	endMainLoop												:	BOOL;					// End of main loop reached
	endSubLoop												:	BOOL;					// End of sub loop reached                                              
	ElementCount											:	DINT;					// No of array elements
	stackCount,left,right,i,j,k								:	DINT;					// running variables 	
	stack													:	ARRAY[1..32] OF UDINT;	// stack size 32 => ~1 Mio elements *)	
	                                					
	pElement_1												:	POINTER TO BYTE;		// Copy Pointer 1		
	pElement_2												:	POINTER TO BYTE;		// Copy Pointer 2
END_VAR
// ends with true in case of no error	                                    					 					
IF SizeOfStruct = 0 OR SizeOfData = 0
	OR pData = 0 OR pCompareElement = 0
THEN               					                                   					
	bySTRING												:= FALSE;
	RETURN;   
ELSE
	bySTRING												:= TRUE;                          					
END_IF                                 					
          
// calculate no. of Elements                                
ElementCount												:= TO_DINT(SizeOfData / SizeOfStruct);   
                              					
// Quicksort                            					
// initial value of array size          					
left 														:= 1;				// first element
right 														:= ElementCount;	// last element 
stackCount 													:= 1;				// running variable 
                                        	
WHILE NOT endMainLoop DO							
	IF left < right THEN                	
		pPivotElement										:= pCompareElement + (SizeOfStruct * TO_UDINT(SHR(right+left,1)));
		i 													:= left -1;
		j 													:= right +1;
		endSubLoop 											:= FALSE;
		REPEAT
			IF SortInverse
			THEN	// sort descending	
				REPEAT	
					i 										:= i+1;	
					pCmpElement								:= pCompareElement + (SizeOfStruct * TO_UDINT(i-1));
					FOR k := 1 TO MAX_STRING_LENGTH DO // Find unequal char
						// element 1,2 to upper char 	https://www.uni-due.de/hummell/infos/ascii/
						IF pCmpElement^[k] = 0 
							AND IgnoreBlank
						THEN
							CompareElement					:= 127;
						ELSE
							CompareElement					:= SEL(pCmpElement^[k] >= 97(*a*)	AND_THEN pCmpElement^[k] <= 122(*z*), 	pCmpElement^[k],pCmpElement^[k] - 32);		// a --> A
						END_IF						
						IF pPivotElement^[k] = 0 
							AND IgnoreBlank
						THEN
							PivotElement					:= 127;
						ELSE
							PivotElement					:= SEL(pPivotElement^[k] >= 97(*a*) AND_THEN pPivotElement^[k] <= 122(*z*), pPivotElement^[k], 	pPivotElement^[k] - 32);// a --> A
						END_IF
						// Find unequal char
						IF CompareElement <> PivotElement
							OR CompareElement = 0
							OR PivotElement = 0
						THEN
							EXIT;
						END_IF
					END_FOR
				UNTIL (CompareElement <= PivotElement) OR NOT (i < right)	END_REPEAT	
				REPEAT	
					j 										:= j-1;	
					pCmpElement								:= pCompareElement + (SizeOfStruct * TO_UDINT(j-1));
					FOR k := 0 TO MAX_STRING_LENGTH DO // Find unequal char
						// element 1,2 to upper char 	https://www.uni-due.de/hummell/infos/ascii/
						IF pCmpElement^[k] = 0 
							AND IgnoreBlank
						THEN
							CompareElement					:= 127;
						ELSE
							CompareElement					:= SEL(pCmpElement^[k] >= 97(*a*)	AND_THEN pCmpElement^[k] <= 122(*z*), 	pCmpElement^[k],pCmpElement^[k] - 32);		// a --> A
						END_IF
						IF pPivotElement^[k] = 0 
							AND IgnoreBlank
						THEN
							PivotElement					:= 127;
						ELSE
							PivotElement					:= SEL(pPivotElement^[k] >= 97(*a*) AND_THEN pPivotElement^[k] <= 122(*z*), pPivotElement^[k], 	pPivotElement^[k] - 32);// a --> A
						END_IF
						// Find unequal char
						IF CompareElement <> PivotElement
							OR CompareElement = 0
							OR PivotElement = 0
						THEN
							EXIT;
						END_IF
					END_FOR
				UNTIL (CompareElement >= PivotElement) OR NOT (j > left)	END_REPEAT		
			ELSE	// sort ascending
				REPEAT	
					i 										:= i+1;
					pCmpElement								:= pCompareElement + (SizeOfStruct * TO_UDINT(i-1));
					FOR k := 0 TO MAX_STRING_LENGTH DO // Find unequal char
						// element 1,2 to upper char 	https://www.uni-due.de/hummell/infos/ascii/
						IF pCmpElement^[k] = 0 
							AND IgnoreBlank
						THEN
							CompareElement					:= 127;
						ELSE
							CompareElement					:= SEL(pCmpElement^[k] >= 97(*a*)	AND_THEN pCmpElement^[k] <= 122(*z*), 	pCmpElement^[k],pCmpElement^[k] - 32);		// a --> A
						END_IF
						IF pPivotElement^[k] = 0 
							AND IgnoreBlank
						THEN
							PivotElement					:= 127;
						ELSE
							PivotElement					:= SEL(pPivotElement^[k] >= 97(*a*) AND_THEN pPivotElement^[k] <= 122(*z*), pPivotElement^[k], 	pPivotElement^[k] - 32);// a --> A
						END_IF
						// Find unequal char
						IF CompareElement <> PivotElement
							OR CompareElement = 0
							OR PivotElement = 0
						THEN
							EXIT;
						END_IF
					END_FOR
				UNTIL (CompareElement >= PivotElement)	OR NOT (i < right)	END_REPEAT;				
				REPEAT	
					j 										:= j-1;	
					pCmpElement								:= pCompareElement + (SizeOfStruct * TO_UDINT(j-1));
					FOR k := 0 TO MAX_STRING_LENGTH DO // Find unequal char
						// element 1,2 to upper char 	https://www.uni-due.de/hummell/infos/ascii/
						IF pCmpElement^[k] = 0 
							AND IgnoreBlank
						THEN	
							CompareElement					:= 127;
						ELSE
							CompareElement					:= SEL(pCmpElement^[k] >= 97(*a*)	AND_THEN pCmpElement^[k] <= 122(*z*), 	pCmpElement^[k],pCmpElement^[k] - 32);		// a --> A
						END_IF
						IF pPivotElement^[k] = 0
							AND IgnoreBlank 
						THEN
							PivotElement					:= 127;
						ELSE
							PivotElement					:= SEL(pPivotElement^[k] >= 97(*a*) AND_THEN pPivotElement^[k] <= 122(*z*), pPivotElement^[k], 	pPivotElement^[k] - 32);// a --> A
						END_IF
						// Find unequal char
						IF CompareElement <> PivotElement
							OR CompareElement = 0
							OR PivotElement = 0
						THEN
							EXIT;
						END_IF
					END_FOR
				UNTIL (CompareElement <= PivotElement) OR NOT (j > left)	END_REPEAT;
			END_IF
			IF i >= j THEN
				endSubLoop									:= TRUE;
			ELSE                    					
				Allocate(SizeOfStruct);
				pElement_1									:= pData + (SizeOfStruct * TO_UDINT(j-1));
				pElement_2									:= pData + (SizeOfStruct * TO_UDINT(i-1));
				
				IF pElement_Tmp = 0 
					OR_ELSE MEMCPY(pElement_Tmp, pElement_1,	SizeOfStruct) = 0
					OR_ELSE MEMCPY(pElement_1,	pElement_2,		SizeOfStruct) = 0
					OR_ELSE MEMCPY(pElement_2,	pElement_Tmp,	SizeOfStruct) = 0
				THEN
					bySTRING								:= FALSE;
					RETURN;	
				END_IF

			END_IF
		UNTIL endSubLoop END_REPEAT;		
		stack[stackCount] 									:= TO_UDINT(right); 	// save right in stack			
		IF stackCount < 32              					
		THEN                            					
			stackCount 										:= stackCount +1;
		ELSE															// Error stack Limit    
			endMainLoop 									:= TRUE;
			bySTRING										:= FALSE;			
		END_IF                          					
		right 												:= MAX(left, i-1);
	ELSE                                
		IF stackCount = 1 THEN          
			endMainLoop 									:= TRUE;
		ELSE                            					
			left 											:= right+1;       
			stackCount 										:= stackCount -1;	// load from stack
			right											:= TO_DINT(stack[stackCount]);
		END_IF
	END_IF
END_WHILE
END_METHOD

METHOD byTIME : BOOL // returns true if sort ends successfully 
VAR_INPUT
	pData													: 	POINTER TO BYTE := 0;	// ADR(Array) 	
	SizeOfData												: 	UDINT := 0;				// SIZEOF(Array)
	pCompareElement											: 	POINTER TO BYTE := 0;	// ADR(Array[1].TIME)		
	SizeOfStruct											: 	UDINT := 0;				// SIZEOF(Array[1]) 	
END_VAR                                                 
VAR        
	pPivotElement											: 	POINTER TO TIME;		// Pivot value
	PivotElement											: 	TIME;					// Pivot value as TIME	
	pCmpElement												:	POINTER TO TIME;		// compare value
	                                					                            	
	endMainLoop												:	BOOL;					// End of main loop reached
	endSubLoop												:	BOOL;					// End of sub loop reached                                              
	ElementCount											:	DINT;					// No of array elements
	stackCount,left,right,i,j								:	DINT;					// running variables 	
	stack													:	ARRAY[1..32] OF UDINT;	// stack size 32 => ~1 Mio elements *)	
	                                					
	pElement_1												:	POINTER TO BYTE;		// Copy Pointer 1		
	pElement_2												:	POINTER TO BYTE;		// Copy Pointer 2
END_VAR
// ends with true in case of no error	                                    					 					
IF SizeOfStruct = 0 OR SizeOfData = 0
	OR pData = 0 OR pCompareElement = 0
THEN               					                                   					
	byTIME													:= FALSE;
	RETURN;   
ELSE
	byTIME													:= TRUE;                          					
END_IF   

// calculate no. of Elements                                
ElementCount												:= TO_DINT(SizeOfData / SizeOfStruct);                                   					
                                        					
// Quicksort                            					
// initial value of array size          					
left 														:= 1;				// first element
right 														:= ElementCount;	// last element 
stackCount 													:= 1;				// running variable 
                                        	
WHILE NOT endMainLoop DO							
	IF left < right THEN                	
		pPivotElement										:= pCompareElement + (SizeOfStruct * TO_UDINT(SHR(right+left,1)));
		PivotElement										:= pPivotElement^;
		i 													:= left -1;
		j 													:= right +1;
		endSubLoop 											:= FALSE;
		REPEAT
			IF SortInverse
			THEN	// sort descending	
				REPEAT	
					i 										:= i+1;	
					pCmpElement								:= pCompareElement + (SizeOfStruct * TO_UDINT(i-1));
				UNTIL (pCmpElement^ <= PivotElement) OR NOT (i < right)	END_REPEAT	
				REPEAT	
					j 										:= j-1;	
					pCmpElement								:= pCompareElement + (SizeOfStruct * TO_UDINT(j-1));
				UNTIL (pCmpElement^ >= PivotElement) OR NOT (j > left)	END_REPEAT		
			ELSE	// sort ascending
				REPEAT	
					i 										:= i+1;
					pCmpElement								:= pCompareElement + (SizeOfStruct * TO_UDINT(i-1));
				UNTIL (pCmpElement^ >= PivotElement)	OR NOT (i < right)	END_REPEAT;				
				REPEAT	
					j 										:= j-1;	
					pCmpElement								:= pCompareElement + (SizeOfStruct * TO_UDINT(j-1));
				UNTIL (pCmpElement^ <= PivotElement) OR NOT (j > left)	END_REPEAT;
			END_IF
			IF i >= j THEN
				endSubLoop									:= TRUE;
			ELSE                    					
				Allocate(SizeOfStruct);
				pElement_1									:= pData + (SizeOfStruct * TO_UDINT(j-1));
				pElement_2									:= pData + (SizeOfStruct * TO_UDINT(i-1));
				
				IF pElement_Tmp = 0 
					OR_ELSE MEMCPY(pElement_Tmp, pElement_1,	SizeOfStruct) = 0
					OR_ELSE MEMCPY(pElement_1,	pElement_2,		SizeOfStruct) = 0
					OR_ELSE MEMCPY(pElement_2,	pElement_Tmp,	SizeOfStruct) = 0
				THEN
					byTIME									:= FALSE;
					RETURN;	
				END_IF

			END_IF
		UNTIL endSubLoop END_REPEAT;		
		stack[stackCount] 									:= TO_UDINT(right); 	// save right in stack			
		IF stackCount < 32              					
		THEN                            					
			stackCount 										:= stackCount +1;
		ELSE															// Error stack Limit    
			endMainLoop 									:= TRUE;
			byTIME											:= FALSE;			
		END_IF                          					
		right 												:= MAX(left, i-1);
	ELSE                                
		IF stackCount = 1 THEN          
			endMainLoop 									:= TRUE;
		ELSE                            					
			left 											:= right+1;       
			stackCount 										:= stackCount -1;	// load from stack
			right											:= TO_DINT(stack[stackCount]);
		END_IF
	END_IF
END_WHILE
END_METHOD

METHOD byUINT : BOOL // returns true if sort ends successfully 
VAR_INPUT
	pData													: 	POINTER TO BYTE := 0;	// ADR(Array) 	
	SizeOfData												: 	UDINT := 0;				// SIZEOF(Array)
	pCompareElement											: 	POINTER TO BYTE := 0;	// ADR(Array[1].UINT)		
	SizeOfStruct											: 	UDINT := 0;				// SIZEOF(Array[1]) 	
END_VAR                                                 
VAR        
	pPivotElement											: 	POINTER TO UINT;		// Pivot value	
	PivotElement											: 	UINT;					// Pivot value as UINT	
	pCmpElement												:	POINTER TO UINT;		// compare value
	                                					                            	
	endMainLoop												:	BOOL;					// End of main loop reached
	endSubLoop												:	BOOL;					// End of sub loop reached                                              
	ElementCount											:	DINT;					// No of array elements
	stackCount,left,right,i,j								:	DINT;					// running variables 	
	stack													:	ARRAY[1..32] OF UDINT;	// stack size 32 => ~1 Mio elements *)	
	                                					
	pElement_1												:	POINTER TO BYTE;		// Copy Pointer 1		
	pElement_2												:	POINTER TO BYTE;		// Copy Pointer 2
END_VAR
// ends with true in case of no error	                                    					 					
IF SizeOfStruct = 0 OR SizeOfData = 0
	OR pData = 0 OR pCompareElement = 0
THEN               					                                   					
	byUINT													:= FALSE;
	RETURN;   
ELSE
	byUINT													:= TRUE;                          					
END_IF     

// calculate no. of Elements                                
ElementCount												:= TO_DINT(SizeOfData / SizeOfStruct);                                 					
                                        					
// Quicksort                            					
// initial value of array size          					
left 														:= 1;				// first element
right 														:= ElementCount;	// last element 
stackCount 													:= 1;				// running variable 
                                        	
WHILE NOT endMainLoop DO							
	IF left < right THEN                	
		pPivotElement										:= pCompareElement + (SizeOfStruct * TO_UDINT(SHR(right+left,1)));
		PivotElement										:= pPivotElement^;
		i 													:= left -1;
		j 													:= right +1;
		endSubLoop 											:= FALSE;
		REPEAT
			IF SortInverse
			THEN	// sort descending	
				REPEAT	
					i 										:= i+1;	
					pCmpElement								:= pCompareElement + (SizeOfStruct * TO_UDINT(i-1));
				UNTIL (pCmpElement^ <= PivotElement) OR NOT (i < right)	END_REPEAT	
				REPEAT	
					j 										:= j-1;	
					pCmpElement								:= pCompareElement + (SizeOfStruct * TO_UDINT(j-1));
				UNTIL (pCmpElement^ >= PivotElement) OR NOT (j > left)	END_REPEAT		
			ELSE	// sort ascending
				REPEAT	
					i 										:= i+1;
					pCmpElement								:= pCompareElement + (SizeOfStruct * TO_UDINT(i-1));
				UNTIL (pCmpElement^ >= PivotElement)	OR NOT (i < right)	END_REPEAT;				
				REPEAT	
					j 										:= j-1;	
					pCmpElement								:= pCompareElement + (SizeOfStruct * TO_UDINT(j-1));
				UNTIL (pCmpElement^ <= PivotElement) OR NOT (j > left)	END_REPEAT;
			END_IF
			IF i >= j THEN
				endSubLoop									:= TRUE;
			ELSE                    					
				Allocate(SizeOfStruct);
				pElement_1									:= pData + (SizeOfStruct * TO_UDINT(j-1));
				pElement_2									:= pData + (SizeOfStruct * TO_UDINT(i-1));
				
				IF pElement_Tmp = 0 
					OR_ELSE MEMCPY(pElement_Tmp, pElement_1,	SizeOfStruct) = 0
					OR_ELSE MEMCPY(pElement_1,	pElement_2,		SizeOfStruct) = 0
					OR_ELSE MEMCPY(pElement_2,	pElement_Tmp,	SizeOfStruct) = 0
				THEN
					byUINT									:= FALSE;
					RETURN;	
				END_IF

			END_IF
		UNTIL endSubLoop END_REPEAT;		
		stack[stackCount] 									:= TO_UDINT(right); 	// save right in stack			
		IF stackCount < 32              					
		THEN                            					
			stackCount 										:= stackCount +1;
		ELSE															// Error stack Limit    
			endMainLoop 									:= TRUE;
			byUINT											:= FALSE;			
		END_IF                          					
		right 												:= MAX(left, i-1);
	ELSE                                
		IF stackCount = 1 THEN          
			endMainLoop 									:= TRUE;
		ELSE                            					
			left 											:= right+1;       
			stackCount 										:= stackCount -1;	// load from stack
			right											:= TO_DINT(stack[stackCount]);
		END_IF
	END_IF
END_WHILE
END_METHOD

METHOD byUSINT : BOOL // returns true if sort ends successfully 
VAR_INPUT
	pData													: 	POINTER TO BYTE := 0;	// ADR(Array) 	
	SizeOfData												: 	UDINT := 0;				// SIZEOF(Array)
	pCompareElement											: 	POINTER TO BYTE := 0;	// ADR(Array[1].USINT)		
	SizeOfStruct											: 	UDINT := 0;				// SIZEOF(Array[1]) 	
END_VAR                                                 
VAR        
	pPivotElement											: 	POINTER TO USINT;		// Pivot value	
	PivotElement											: 	USINT;					// Pivot value as USINT
	pCmpElement												:	POINTER TO USINT;		// compare value
	                                					                            	
	endMainLoop												:	BOOL;					// End of main loop reached
	endSubLoop												:	BOOL;					// End of sub loop reached                                              
	ElementCount											:	DINT;					// No of array elements
	stackCount,left,right,i,j								:	DINT;					// running variables 	
	stack													:	ARRAY[1..32] OF UDINT;	// stack size 32 => ~1 Mio elements *)	
	                                					
	pElement_1												:	POINTER TO BYTE;		// Copy Pointer 1		
	pElement_2												:	POINTER TO BYTE;		// Copy Pointer 2
END_VAR
// ends with true in case of no error	                                    					 					
IF SizeOfStruct = 0 OR SizeOfData = 0
	OR pData = 0 OR pCompareElement = 0
THEN               					                                   					
	byUSINT													:= FALSE;
	RETURN;   
ELSE
	byUSINT													:= TRUE;                          					
END_IF    

// calculate no. of Elements                                
ElementCount												:= TO_DINT(SizeOfData / SizeOfStruct);                               					
                                        					
// Quicksort                            					
// initial value of array size          					
left 														:= 1;				// first element
right 														:= ElementCount;	// last element 
stackCount 													:= 1;				// running variable 
                                        	
WHILE NOT endMainLoop DO							
	IF left < right THEN                	
		pPivotElement										:= pCompareElement + (SizeOfStruct * TO_UDINT(SHR(right+left,1)));
		PivotElement										:= pPivotElement^;
		i 													:= left -1;
		j 													:= right +1;
		endSubLoop 											:= FALSE;
		REPEAT
			IF SortInverse
			THEN	// sort descending	
				REPEAT	
					i 										:= i+1;	
					pCmpElement								:= pCompareElement + (SizeOfStruct * TO_UDINT(i-1));
				UNTIL (pCmpElement^ <= PivotElement) OR NOT (i < right)	END_REPEAT	
				REPEAT	
					j 										:= j-1;	
					pCmpElement								:= pCompareElement + (SizeOfStruct * TO_UDINT(j-1));
				UNTIL (pCmpElement^ >= PivotElement) OR NOT (j > left)	END_REPEAT		
			ELSE	// sort ascending
				REPEAT	
					i 										:= i+1;
					pCmpElement								:= pCompareElement + (SizeOfStruct * TO_UDINT(i-1));
				UNTIL (pCmpElement^ >= PivotElement)	OR NOT (i < right)	END_REPEAT;				
				REPEAT	
					j 										:= j-1;	
					pCmpElement								:= pCompareElement + (SizeOfStruct * TO_UDINT(j-1));
				UNTIL (pCmpElement^ <= PivotElement) OR NOT (j > left)	END_REPEAT;
			END_IF
			IF i >= j THEN
				endSubLoop									:= TRUE;
			ELSE                    					
				Allocate(SizeOfStruct);
				pElement_1									:= pData + (SizeOfStruct * TO_UDINT(j-1));
				pElement_2									:= pData + (SizeOfStruct * TO_UDINT(i-1));
				
				IF pElement_Tmp = 0 
					OR_ELSE MEMCPY(pElement_Tmp, pElement_1,	SizeOfStruct) = 0
					OR_ELSE MEMCPY(pElement_1,	pElement_2,		SizeOfStruct) = 0
					OR_ELSE MEMCPY(pElement_2,	pElement_Tmp,	SizeOfStruct) = 0
				THEN
					byUSINT									:= FALSE;
					RETURN;	
				END_IF

			END_IF
		UNTIL endSubLoop END_REPEAT;		
		stack[stackCount] 									:= TO_UDINT(right); 	// save right in stack			
		IF stackCount < 32              					
		THEN                            					
			stackCount 										:= stackCount +1;
		ELSE															// Error stack Limit    
			endMainLoop 									:= TRUE;
			byUSINT											:= FALSE;			
		END_IF                          					
		right 												:= MAX(left, i-1);
	ELSE                                
		IF stackCount = 1 THEN          
			endMainLoop 									:= TRUE;
		ELSE                            					
			left 											:= right+1;       
			stackCount 										:= stackCount -1;	// load from stack
			right											:= TO_DINT(stack[stackCount]);
		END_IF
	END_IF
END_WHILE
END_METHOD

METHOD byWSTRING : BOOL // returns true if sort ends successfully 
VAR_INPUT
	pData													: 	POINTER TO BYTE := 0;	// ADR(Array) 	
	SizeOfData												: 	UDINT := 0;				// SIZEOF(Array)
	pCompareElement											: 	POINTER TO BYTE := 0;	// ADR(Array[1].WSTRING)		
	SizeOfStruct											: 	UDINT := 0;				// SIZEOF(Array[1]) 	
END_VAR                                                                                            
VAR        
	pPivotElement											: 	POINTER TO WSTRING(MAX_WSTRING_LENGTH);	// Pivot value	
	pCmpElement												:	POINTER TO WSTRING(MAX_WSTRING_LENGTH);	// compare value
	PivotElement											:	WORD; 					// Pivot value	
	CompareElement											:	WORD; 					// compare value
	                                					                            	
	endMainLoop												:	BOOL;					// End of main loop reached
	endSubLoop												:	BOOL;					// End of sub loop reached                                              
	ElementCount											:	DINT;					// No of array elements
	stackCount,left,right,i,j,k								:	DINT;					// running variables 	
	stack													:	ARRAY[1..32] OF UDINT;	// stack size 32 => ~1 Mio elements *)	
	                                					
	pElement_1												:	POINTER TO BYTE;		// Copy Pointer 1		
	pElement_2												:	POINTER TO BYTE;		// Copy Pointer 2
END_VAR
// ends with true in case of no error	                                    					 					
IF SizeOfStruct = 0 OR SizeOfData = 0
	OR pData = 0 OR pCompareElement = 0
THEN               					                                   					
	byWSTRING												:= FALSE;
	RETURN;   
ELSE
	byWSTRING												:= TRUE;                          					
END_IF                                   					
            
// calculate no. of Elements                                
ElementCount												:= TO_DINT(SizeOfData / SizeOfStruct);   
                            					
// Quicksort                            					
// initial value of array size          					
left 														:= 1;				// first element
right 														:= ElementCount;	// last element 
stackCount 													:= 1;				// running variable 
                                        	
WHILE NOT endMainLoop DO							
	IF left < right THEN                	
		pPivotElement										:= pCompareElement + (SizeOfStruct * TO_UDINT(SHR(right+left,1)));
		i 													:= left -1;
		j 													:= right +1;
		endSubLoop 											:= FALSE;
		REPEAT
			IF SortInverse
			THEN	// sort descending	
				REPEAT	
					i 										:= i+1;	
					pCmpElement								:= pCompareElement + (SizeOfStruct * TO_UDINT(i-1));
					FOR k := 0 TO MAX_WSTRING_LENGTH DO // Find unequal char
						// element 1,2 to upper char 	https://www.uni-due.de/hummell/infos/ascii/
						IF pCmpElement^[k] = 0 
							AND IgnoreBlank
						THEN
							CompareElement					:= 127;
						ELSE
							CompareElement					:= SEL(pCmpElement^[k] >= 97(*a*)	AND_THEN pCmpElement^[k] <= 122(*z*), 	pCmpElement^[k],pCmpElement^[k] - 32);		// a --> A
						END_IF
						IF pPivotElement^[k] = 0 
							AND IgnoreBlank
						THEN
							PivotElement					:= 127;
						ELSE
							PivotElement					:= SEL(pPivotElement^[k] >= 97(*a*) AND_THEN pPivotElement^[k] <= 122(*z*), pPivotElement^[k], 	pPivotElement^[k] - 32);// a --> A
						END_IF
						// Find unequal char
						IF CompareElement <> PivotElement
							OR CompareElement = 0
							OR PivotElement = 0
						THEN
							EXIT;
						END_IF
					END_FOR
				UNTIL (CompareElement <= PivotElement) OR NOT (i < right)	END_REPEAT	
				REPEAT	
					j 										:= j-1;	
					pCmpElement								:= pCompareElement + (SizeOfStruct * TO_UDINT(j-1));
					FOR k := 0 TO MAX_WSTRING_LENGTH DO // Find unequal char
						// element 1,2 to upper char 	https://www.uni-due.de/hummell/infos/ascii/
						IF pCmpElement^[k] = 0 
							AND IgnoreBlank
						THEN
							CompareElement					:= 127;
						ELSE
							CompareElement					:= SEL(pCmpElement^[k] >= 97(*a*)	AND_THEN pCmpElement^[k] <= 122(*z*), 	pCmpElement^[k],pCmpElement^[k] - 32);		// a --> A
						END_IF
						IF pPivotElement^[k] = 0 
							AND IgnoreBlank
						THEN
							PivotElement					:= 127;
						ELSE
							PivotElement					:= SEL(pPivotElement^[k] >= 97(*a*) AND_THEN pPivotElement^[k] <= 122(*z*), pPivotElement^[k], 	pPivotElement^[k] - 32);// a --> A
						END_IF
						// Find unequal char
						IF CompareElement <> PivotElement
							OR CompareElement = 0
							OR PivotElement = 0
						THEN
							EXIT;
						END_IF
					END_FOR
				UNTIL (CompareElement >= PivotElement) OR NOT (j > left)	END_REPEAT		
			ELSE	// sort ascending
				REPEAT	
					i 										:= i+1;
					pCmpElement								:= pCompareElement + (SizeOfStruct * TO_UDINT(i-1));
					FOR k := 0 TO MAX_WSTRING_LENGTH DO // Find unequal char
						// element 1,2 to upper char 	https://www.uni-due.de/hummell/infos/ascii/
						IF pCmpElement^[k] = 0 
							AND IgnoreBlank
						THEN
							CompareElement					:= 127;
						ELSE
							CompareElement					:= SEL(pCmpElement^[k] >= 97(*a*)	AND_THEN pCmpElement^[k] <= 122(*z*), 	pCmpElement^[k],pCmpElement^[k] - 32);		// a --> A
						END_IF
						IF pPivotElement^[k] = 0 
							AND IgnoreBlank
						THEN
							PivotElement					:= 127;
						ELSE
							PivotElement					:= SEL(pPivotElement^[k] >= 97(*a*) AND_THEN pPivotElement^[k] <= 122(*z*), pPivotElement^[k], 	pPivotElement^[k] - 32);// a --> A
						END_IF
						// Find unequal char
						IF CompareElement <> PivotElement
							OR CompareElement = 0
							OR PivotElement = 0
						THEN
							EXIT;
						END_IF
					END_FOR
				UNTIL (CompareElement >= PivotElement)	OR NOT (i < right)	END_REPEAT;				
				REPEAT	
					j 										:= j-1;	
					pCmpElement								:= pCompareElement + (SizeOfStruct * TO_UDINT(j-1));
					FOR k := 0 TO MAX_WSTRING_LENGTH DO // Find unequal char
						// element 1,2 to upper char 	https://www.uni-due.de/hummell/infos/ascii/
						IF pCmpElement^[k] = 0 
							AND IgnoreBlank
						THEN
							CompareElement					:= 127;
						ELSE
							CompareElement					:= SEL(pCmpElement^[k] >= 97(*a*)	AND_THEN pCmpElement^[k] <= 122(*z*), 	pCmpElement^[k],pCmpElement^[k] - 32);		// a --> A
						END_IF
						IF pPivotElement^[k] = 0 
							AND IgnoreBlank
						THEN
							PivotElement					:= 127;
						ELSE
							PivotElement					:= SEL(pPivotElement^[k] >= 97(*a*) AND_THEN pPivotElement^[k] <= 122(*z*), pPivotElement^[k], 	pPivotElement^[k] - 32);// a --> A
						END_IF
						// Find unequal char
						IF CompareElement <> PivotElement
							OR CompareElement = 0
							OR PivotElement = 0
						THEN
							EXIT;
						END_IF
					END_FOR
				UNTIL (CompareElement <= PivotElement) OR NOT (j > left)	END_REPEAT;
			END_IF
			IF i >= j THEN
				endSubLoop									:= TRUE;
			ELSE                    					
				Allocate(SizeOfStruct);
				pElement_1									:= pData + (SizeOfStruct * TO_UDINT(j-1));
				pElement_2									:= pData + (SizeOfStruct * TO_UDINT(i-1));
				
				IF pElement_Tmp = 0 
					OR_ELSE MEMCPY(pElement_Tmp, pElement_1,	SizeOfStruct) = 0
					OR_ELSE MEMCPY(pElement_1,	pElement_2,		SizeOfStruct) = 0
					OR_ELSE MEMCPY(pElement_2,	pElement_Tmp,	SizeOfStruct) = 0
				THEN
					byWSTRING								:= FALSE;
					RETURN;	
				END_IF

			END_IF
		UNTIL endSubLoop END_REPEAT;		
		stack[stackCount] 									:= TO_UDINT(right); 	// save right in stack			
		IF stackCount < 32              					
		THEN                            					
			stackCount 										:= stackCount +1;
		ELSE															// Error stack Limit    
			endMainLoop 									:= TRUE;
			byWSTRING										:= FALSE;			
		END_IF                          					
		right 												:= MAX(left, i-1);
	ELSE                                
		IF stackCount = 1 THEN          
			endMainLoop 									:= TRUE;
		ELSE                            					
			left 											:= right+1;       
			stackCount 										:= stackCount -1;	// load from stack
			right											:= TO_DINT(stack[stackCount]);
		END_IF
	END_IF
END_WHILE
END_METHOD

METHOD FB_exit : BOOL
VAR_INPUT
	bInCopyCode : BOOL; // if TRUE, the exit method is called for exiting an instance that is copied afterwards (online change).
END_VAR
IF NOT bInCopyCode AND pElement_Tmp <> 0
THEN //Release memory in case the PLC stopps
	__DELETE(pElement_Tmp);
END_IF
END_METHOD

END_FUNCTION_BLOCK

// ---- POUs/DataBuffer/Ringbuffer/Ringbuffer.TcPOU
//Ringbuffer based on external memory
FUNCTION_BLOCK Ringbuffer EXTENDS RingbufferBase
VAR_INPUT	
END_VAR
VAR_OUTPUT
END_VAR    
VAR
END_VAR

METHOD PUBLIC dequeue : BOOL //TRUE if method was successful
VAR_INPUT
	pData													: 	POINTER TO BYTE ;
	SizeOfData												: 	UDINT ;
	pMemory													: 	POINTER TO BYTE ;
	SizeOfMemory											: 	UDINT ;
END_VAR
Dequeue := SUPER^._Dequeue(pData,SizeOfData,pMemory,SizeOfMemory);
END_METHOD

METHOD PUBLIC dequeueStream : BOOL //TRUE if method was successful
VAR_INPUT
	pData													: 	POINTER TO BYTE ;
	SizeOfStream											:	UDINT ; //n * Size of last entry and not greater than SizeOfMemory
	pMemory													: 	POINTER TO BYTE;
	SizeOfMemory											: 	UDINT ;
END_VAR
VAR
END_VAR
DequeueStream := SUPER^._DequeueStream(pData,SizeOfStream,pMemory,SizeOfMemory);
END_METHOD

METHOD PUBLIC enqueue : BOOL //TRUE if method was successful
VAR_INPUT
	pData													: 	POINTER TO BYTE ;
	SizeOfData												: 	UDINT ;
	pMemory													: 	POINTER TO BYTE ;
	SizeOfMemory											: 	UDINT ;
END_VAR
Enqueue := SUPER^._Enqueue(pData,SizeOfData,pMemory,SizeOfMemory);
END_METHOD

METHOD PUBLIC enqueueStream : BOOL
VAR_INPUT
	pData													: 	POINTER TO BYTE ;
	SizeOfData												: 	UDINT ; //Size of one entry
	SizeOfStream											:	UDINT ; //n * SizeofData and not greater than SizeOfMemory
	pMemory													: 	POINTER TO BYTE ;
	SizeOfMemory											: 	UDINT ;
END_VAR
VAR
END_VAR
EnqueueStream := SUPER^._EnqueueStream(pData,SizeOfData,SizeOfStream,pMemory,SizeOfMemory);
END_METHOD

//Reset complete ring buffer
METHOD PUBLIC reset : BOOL //TRUE if method is finnished
VAR_INPUT
	pMemory													: 	POINTER TO BYTE := 0;
	SizeOfMemory											: 	UDINT := 0;
END_VAR
reset := SUPER^._reset(pMemory,SizeOfMemory);
END_METHOD

END_FUNCTION_BLOCK

// ---- POUs/DataBuffer/Ringbuffer/RingbufferCharSimple.TcPOU
//Ringbuffer with a internal char array (String) for a simple num list implementation
FUNCTION_BLOCK RingbufferCharSimple EXTENDS RingbufferBase
VAR_OUTPUT CONSTANT
	MIN_BUFFER												:	UDINT := 0; //Default min index of string 
	MAX_BUFFER												:	UDINT := PARAM.RINGBUFFER_CHAR_SIMPLE_MAX_BUFFER; //Ringbuffer buffer end index - see library parameter to customize parameter
END_VAR   
VAR_INPUT
END_VAR
VAR_OUTPUT
	Buffer													:	STRING[MAX_BUFFER]; //Char buffer 
END_VAR
VAR
END_VAR

;

METHOD PUBLIC dequeue : BOOL //TRUE if method was successful
VAR_IN_OUT
	value													: BYTE;	
END_VAR
Dequeue := SUPER^._Dequeue(ADR(Value),SizeOfEntry,ADR(Buffer),SIZEOF(Buffer));
END_METHOD

METHOD PUBLIC dequeueStream : BOOL //TRUE if method was successful
VAR_INPUT
	pData													:	POINTER TO BYTE;
	SizeOfStream											:	UDINT ; //Not greater than SizeOfMemory
END_VAR
DequeueStream := SUPER^._DequeueStream(pData, SizeOfStream,  ADR(Buffer),TO_UDINT(MAX_BUFFER));
END_METHOD

METHOD PUBLIC enqueue : BOOL //TRUE if method was successful
VAR_INPUT
	Value													:	BYTE;
END_VAR
Enqueue := SUPER^._Enqueue(ADR(Value),SIZEOF(Value),ADR(Buffer),SIZEOF(Buffer));
END_METHOD

METHOD PUBLIC enqueueStream : BOOL //TRUE if method was successful
VAR_INPUT
	pData													:	POINTER TO BYTE;
	SizeOfStream											:	UDINT ; //Not greater than SizeOfMemory
END_VAR
EnqueueStream := SUPER^._EnqueueStream(pData,SIZEOF(BUFFER[MIN_BUFFER]), SizeOfStream,ADR(Buffer),TO_UDINT(MAX_BUFFER));
END_METHOD

//Reset complete ring buffer
METHOD PUBLIC reset : BOOL //TRUE if method is finnished
VAR_INPUT
END_VAR
reset := SUPER^._reset(ADR(Buffer),SIZEOF(Buffer));
END_METHOD

END_FUNCTION_BLOCK

// ---- POUs/DataBuffer/Ringbuffer/RingbufferByteSimple.TcPOU
//Ringbuffer with a internal Byte array for a simple data buffer implementation 
FUNCTION_BLOCK RingbufferByteSimple EXTENDS RingbufferBase
VAR_OUTPUT CONSTANT
	MIN_BUFFER												:	UDINT := 1; //Ringbuffer start index 
	MAX_BUFFER												:	uDINT := PARAM.RINGBUFFER_BYTE_SIMPLE_MAX_BUFFER; //Ringbuffer buffer end index - see library parameter to customize parameter
END_VAR   
VAR_INPUT
END_VAR
VAR_OUTPUT
	Buffer													:	ARRAY[MIN_BUFFER..MAX_BUFFER] OF BYTE; //Byte buffer 
END_VAR
VAR 
END_VAR

;

METHOD PUBLIC dequeue : BOOL //TRUE if method was successful
VAR_IN_OUT
	value													: BYTE;	
END_VAR
IF TestAndSet(Interlock)
THEN	
	IF Count > 0
	THEN 
		(* copy dataset *)		
		ReadIdx												:= ReadIdx + 1;
		IF (ReadIdx) > MAX_BUFFER
		THEN
			ReadIdx											:= TO_UDINT(MIN_BUFFER);				
		END_IF
		
		Value												:= Buffer[ReadIdx];
		
		Count 												:= MAX(0,Count - 1);
		Empty 												:= Count = 0;
		Full												:= FALSE;
		Dequeue												:= TRUE;	
	ELSE 
		Dequeue												:= FALSE;
	END_IF
	
	Interlock												:= FALSE;
ELSE
	Dequeue													:= FALSE;
END_IF
END_METHOD

METHOD PUBLIC dequeueStream : BOOL //TRUE if method was successful
VAR_INPUT
	pData													:	POINTER TO BYTE;
	SizeOfStream											:	UDINT;	
END_VAR
DequeueStream := super^._DequeueStream(pData, SizeOfStream,  ADR(Buffer),SIZEOF(Buffer));
END_METHOD

METHOD PUBLIC enqueue : BOOL //TRUE if method was successful
VAR_INPUT
	Value													:	BYTE;
END_VAR
IF TestAndSet(Interlock)
THEN			
	Enqueue													:= FALSE;

	IF Count < MAX_BUFFER OR Overwrite
	THEN
		IF MAX_BUFFER = Count 
		THEN //Adapt read index if write index is in front of read index
			ReadIdx											:= ReadIdx + 1;
			IF ReadIdx > TO_UDINT(MAX_BUFFER)
			THEN
				ReadIdx										:= TO_UDINT(MIN_BUFFER);							
			END_IF
		END_IF		
		WriteIdx											:= WriteIdx + 1;	
		IF WriteIdx > TO_UDINT(MAX_BUFFER)
		THEN
			WriteIdx										:= TO_UDINT(MIN_BUFFER);
		END_IF
	
		Buffer[WriteIdx]									:= Value;
	
		Count												:= MIN(Count + 1,  MAX_BUFFER);
		Full												:= Count >= MAX_BUFFER;
		Empty 												:= FALSE;	
		Enqueue												:= TRUE;
	END_IF
	
	Interlock												:= FALSE;
ELSE
	Enqueue													:= FALSE;
END_IF
END_METHOD

METHOD PUBLIC enqueueStream : BOOL //TRUE if method was successful
VAR_INPUT
	pData													:	POINTER TO BYTE;
	SizeOfStream											:	UDINT;
END_VAR
EnqueueStream := SUPER^._EnqueueStream(pData, SIZEOF(BUFFER[MIN_BUFFER] ), SizeOfStream,ADR(Buffer),SIZEOF(Buffer));
END_METHOD

//Reset complete ring buffer
METHOD PUBLIC reset : BOOL //TRUE if method is finnished
VAR_INPUT
END_VAR
reset := SUPER^._reset(ADR(Buffer),SIZEOF(Buffer));
END_METHOD

END_FUNCTION_BLOCK

// ---- POUs/EventLogger/TriggerEvents/EventHandlingGrp50.TcPOU
{attribute 'no_check'}
//Event group with single source id - for a convenient control of <MAX_EVENTS>
//Each single event handling FB is accessible, so that signal flag, information text and alarm class could be used
FUNCTION_BLOCK EventHandlingGrp50
VAR_OUTPUT CONSTANT
	MIN_EVENT												:	INT := 1; 
	MAX_EVENT												:	INT := 50;
END_VAR                                                 	
VAR_INPUT                                               	
	ConfirmTrig												:	BOOL := FALSE; //Acknowledge event
	SourceId												: 	UDINT := 0; //Source id for all events of this group
	no														:	ARRAY [MIN_EVENT..MAX_EVENT] OF EventHandling; //Array of single event handling FBs 
	Disable													:	BOOL := FALSE; //Disable all events 
	AutoConfirm												:	BOOL := FALSE; //All events will be acknowledged if flag is gone *)
	SetClass												:	E_TcEventClass := TC2_SYSTEM.TCEVENTCLASS_ALARM;// if set class is <> ALARM -> all events set to this Eventclass
	MsgOffset												:	INT := 0; //Offset to change default message id to MIN_EVENT to MsgOffset
END_VAR                                                 	
VAR_OUTPUT    
{attribute 'displaymode':='binary'}
	Status													:	DWORD; (*	.0 - .8 = event of <class id> is active / .15 confirm required / .16 = Level 0 , .17 = Level 1 , .18 = Level 2, ..........
																			TCEVENTCLASS_NONE			:=0,	(* No class *)
																			TCEVENTCLASS_MAINTENANCE	:=1,	(* Maintenance hint *)
																			TCEVENTCLASS_MESSAGE		:=2,	(* Message *)
																			TCEVENTCLASS_HINT			:=3,	(* Hint *)
																			TCEVENTCLASS_STATEINFO		:=4,	(* State information *)
																			TCEVENTCLASS_INSTRUCTION	:=5,	(* Instruction *)
																			TCEVENTCLASS_WARNING		:=6,	(* Warning *)
																			TCEVENTCLASS_ALARM			:=7,	(* Alarm *)
																			TCEVENTCLASS_PARAMERROR		:=8		(* Parameter error *)  *)
	NoOfActiveEvents										:	INT;
END_VAR                                                 	
VAR                                                     	
	_Mem													:	BYTE;
	Disabled												:	BOOL;
	i 														:	INT;
END_VAR

(* EventHandlingGrp			V4.1	*)
(************************************)

(* status ***************************)
Status  													:= 0;
NoOfActiveEvents											:= 0;

IF(Disable OR SourceId = 0)AND Disabled
THEN
	RETURN;
ELSE
	Disabled												:= Disable OR SourceId = 0;
	
	FOR i := MIN_EVENT TO MAX_EVENT 
	DO
		(* Init Default Class *)
		IF SetClass <> TC2_SYSTEM.TCEVENTCLASS_ALARM
			AND NOT _Mem.7
		THEN
			no[i].eClass										:= SetClass;
			_Mem.7											:= i = MAX_EVENT;
		END_IF                                  			
		                                        			
		IF Disable OR SourceId = 0              			
		THEN                                    			
			no[i].Flag 										:= FALSE;
			no[i].ConfirmTrig 								:= no[i].State <> TCEVENTSTATE_INVALID AND no[i].State <> TCEVENTSTATE_RESETCON;
		ELSIF Confirmtrig                             			
		THEN                                    	
			no[i].ConfirmTrig 								:= TRUE;
			_Mem.0 											:= Confirmtrig;
                                                			
		ELSIF _Mem.0                            			
		THEN                                    			
			no[i].ConfirmTrig 								:= FALSE;
			_Mem.0 											:= i <> MAX_EVENT;

		ELSIF AutoConfirm
		THEN
			IF NOT no[i].Flag
				AND no[i].State <> TCEVENTSTATE_INVALID
				AND no[i].State <> TCEVENTSTATE_RESETCON
			THEN
				no[i].ConfirmTrig 							:= TRUE;
			ELSE                                			
				no[i].ConfirmTrig 							:= FALSE;
			END_IF                              			
		END_IF                                  	
                                                	
		(* Mem current Event *)                 	
		IF no[i].State <> TCEVENTSTATE_INVALID OR no[i].Flag 
		THEN
			_Mem.1											:= TRUE;
			(* Call Event *)
			no[i](
				Flag	:= ,
				ConfirmTrig := ,
				MsgId	:= TO_UINT(i + MsgOffset),
				SourceId:= SourceId,
				eClass	:= (* see grp call *),
				Text1	:= (* see grp call *),
				Text2	:= (* see grp call *),
				pText3	:= (* see grp call *),
				State	=> );
		END_IF

		(* Set info flags *)
		IF	no[i].State <> TCEVENTSTATE_INVALID 
		THEN
			NoOfActiveEvents								:= NoOfActiveEvents + 1;
			Status											:= Status OR no[i].Status;
			Disabled										:= FALSE;
		ELSIF _Mem.1
		THEN (* Send one time info event is gone *)
			; 
		END_IF
	END_FOR	
END_IF
(*****************************************************************************************)

METHOD PUBLIC confirm : booL  //Return value = TRUE if execution finished
VAR_INPUT
END_VAR
IF NoOfActiveEvents > 0
THEN
	FOR i := MIN_EVENT TO MAX_EVENT 
	DO
		no[i](ConfirmTrig := TRUE);
	END_FOR
	_Mem.0			:= TRUE;
END_IF

confirm		:= TRUE;
END_METHOD

PROPERTY PUBLIC confirmIsReq : BOOL
GET
confirmIsReq							:= Status.15;
END_GET
END_PROPERTY

PROPERTY PUBLIC isActive : BOOL
GET
IsActive 								:= Status <> 0;
END_GET
END_PROPERTY

END_FUNCTION_BLOCK

// ---- POUs/Fieldbus/CANopen/CANopenMasterDiag.TcPOU
{attribute 'no_check'}
//EL6751 CanOpen Master via EtherCAT
FUNCTION_BLOCK CANopenMasterDiag                   								
VAR_INPUT                   								
	Enable													:	BOOL := TRUE;		//FB will be processed as long as enable is TRUE 
	ConfirmTrig												:	BOOL;               //Resets error with rising edge        								
	SourceId												: 	UDINT :=  103010; 	//Multisource id 
(* Components *)            								
	IO														:	CanOpenMasterIO;
END_VAR                     								
VAR_OUTPUT                  								
	MasterOK												:	BOOL;				//TRUE when Master Device is OK
	FieldOK													:	BOOL;				//TRUE when Field Devices (Slaves) are OK
END_VAR                     	
VAR
(* internal used variables ***********************************************)
	Rx_ErrorCounter											:	USINT := 0;
	Tx_ErrorCounter											: 	USINT := 0;

(* events *********************************************************)
	Event													:	EventHandlingGrp10 := (AutoConfirm	:= FALSE);
	
(* Dummys **********************************************************)
	i														:	INT ;

END_VAR

	(* CanOpen Master Diag Ctrl 					*)
	(************************************************)

(* Work IO *************************************************)
	IO();

(* Events **************************************************)
	IF Event.no[1].Text1 <> IO.Name OR Event.no[1].Text1 <> ''
	THEN
		FOR i := Event.MIN_EVENT TO Event.MAX_EVENT DO
			Event.no[1].Text1								:= IO.Name;
		END_FOR	
	END_IF

(* 
  Bit 0: CAN-Controller is in BUS-OFF
  Bit 1: CAN-Controller warning limit reached
  Bit 2: Rx-Queue overrun
  Bit 3: Hi-Prio Tx-Queue overrun
  Bit 4: Lo-Prio Tx-Queue overrun
  Bit 5: CAN-Send Error
*)
	Event.no[1].Flag 										:= IO.CanState.0;
	Event.no[2].Flag 										:= IO.CanState.1;
	Event.no[3].Flag 										:= IO.CanState.2;   
	Event.no[4].Flag 										:= IO.CanState.3;   
	Event.no[5].Flag 										:= IO.CanState.4; 	
	Event.no[6].Flag 										:= IO.CanState.5;
	
	IF Rx_ErrorCounter <> IO.RXErrorCounter 
	THEN
		Rx_ErrorCounter 									:= IO.RXErrorCounter;
		Event.no[7].Text1 									:= USINT_TO_STRING(Rx_ErrorCounter);
		Event.no[7].Flag									:= TRUE;		
	ELSIF ConfirmTrig
	THEN
		Event.no[7].Flag									:= FALSE;
	END_IF

	IF Tx_ErrorCounter <> IO.TxErrorCounter
	THEN
		Tx_ErrorCounter 									:= IO.TXErrorCounter;
		Event.no[8].Text1 									:= USINT_TO_STRING(Tx_ErrorCounter);
		Event.no[8].Flag									:= TRUE;		
	ELSIF ConfirmTrig
	THEN
		Event.no[8].Flag 									:= FALSE;
	END_IF	

	Event.no[9].Flag 										:= FALSE;
	Event.no[10].Flag 										:= FALSE;	
	
	Event(
		ConfirmTrig := ConfirmTrig,
		Disable		:= NOT Enable,
		SourceId	:= SourceId);
	

(*******************************************************************************************)

END_FUNCTION_BLOCK

// ---- POUs/Fieldbus/EAP/EAP_DEVICE_IO.TcPOU
{attribute 'no_check'}
FUNCTION_BLOCK EAP_DEVICE_IO 
VAR_OUTPUT CONSTANT
END_VAR
VAR_INPUT
	{attribute 'displaymode':='hex'}
	DevCtrl				AT %Q*:	UINT;
END_VAR		
VAR_OUTPUT	
	{attribute 'displaymode':='hex'}
	DevState			AT %I*:	UINT;
	
	LinkError				:	BOOL; //0x0001 = Link error
	IOLockedAfterLinkErr	:	BOOL; //0x0002 = I/O locked after link error (I/O reset required)
	OutOfSendResources		:	BOOL; //0x0010 = Out of send resources (I/O reset required)
	WatchdogTriggered		:	BOOL; //0x0020 = Watchdog triggered
	EthMiniportNotFound		:	BOOL; //0x0040 = Ethernet driver (miniport) not found
	ResetActive				:	BOOL; //0x0080 = I/O reset active
END_VAR
VAR
END_VAR

	(* IOs 									*)
	(****************************************)

(* Read status *****************************************)
	LinkError				:= DevState.0;
	IOLockedAfterLinkErr	:= DevState.1;
	
	OutOfSendResources		:= DevState.4;
	WatchdogTriggered		:= DevState.5;
	EthMiniportNotFound		:= DevState.6;
	ResetActive				:= DevState.7;
	
(*******************************************************)

PROPERTY PUBLIC resetRequired : bool
GET
resetRequired := IOLockedAfterLinkErr or OutOfSendResources;
END_GET
END_PROPERTY

END_FUNCTION_BLOCK

// ---- POUs/Fieldbus/EAP/EAP_SUB_VAR.TcPOU
{attribute 'no_check'}
//Default IOs of a Subscriber network variable 
FUNCTION_BLOCK EAP_SUB_VAR 
VAR_OUTPUT CONSTANT
END_VAR
VAR_INPUT
	VarId					AT %Q*:	UINT;	
	{attribute 'displaymode':='hex'}
	VarCtrl					AT %Q*:	UINT;
END_VAR		
VAR_OUTPUT	
	{attribute 'displaymode':='hex'}
	VarState				AT %I*:	UINT;
	Quality					AT %I*:	UINT;//Duration the variable is not refreshed (in 100µs/0.1ms)	
	CycleIndex				AT %I*:	UINT;//Incremented each publisher cycle
	
	QualityLT					 : LTIME;
	QualityLTMax				 : LTIME;
	
	InvalidHashValueReceived		:	BOOL;
	InvalidVarLengthReceived		:	bool;
END_VAR
VAR
END_VAR

	(* IOs 									*)
	(****************************************)

	QualityLT 								:= TO_LTIME(quality * 100000); //Quality in 100µs to ms
	IF QualityLT > QualityLTMax
	THEN
		QualityLTMax						:= QualityLT;
	END_IF
	
	InvalidHashValueReceived				:= VarState.0;
	InvalidVarLengthReceived				:= VarState.1;

PROPERTY PUBLIC ignoreHashValue : BOOL
GET
ignoreHashValue		:= VarCtrl.0;
END_GET
SET
VarCtrl.0				:= ignoreHashValue;
END_SET
END_PROPERTY

END_FUNCTION_BLOCK

// ---- POUs/Fieldbus/EtherCAT/_Components/EcMasterIO.TcPOU
{attribute 'no_check'}
//EtherCAT Master Device IOs
FUNCTION_BLOCK EcMasterIO
VAR CONSTANT
	DELAY_LINK_OK											:	TIME := T#1S;
END_VAR
VAR_OUTPUT CONSTANT
	MIN_FRAMES												:	INT := 0;
	MAX_FRAMES												:	INT := PARAM.ETHERCAT_MASTER_DEV_IO_MAX_FRAMES; 
END_VAR	            							
VAR_INPUT           							                 							
(* Outputs *)       							
	FrmCtrl											AT %Q*	:	ARRAY [MIN_FRAMES..MAX_FRAMES] OF UINT;	//Link to EtherCAT Master "FrmCtrlXXX" under Outputs, e.g. 0x0001 = prevent 1. EtherCAT command from sending (request NOP)
	FrmWcCtrl										AT %Q*	:	ARRAY [MIN_FRAMES..MAX_FRAMES] OF UINT;	//Link to EtherCAT Master "FrmWcCtrlXXX" under Outputs, e.g. 0x0001 = copy data with wrong working counter of 1. EtherCAT command
	                							
	DevCtrl											AT %Q*	:	UINT := 0; //Link to EtherCAT Master "DevCtrl" under Outputs
END_VAR             							
VAR_OUTPUT          							    
	Name													:	STRING(30) := '';
								
	LinkOK_PortA											:	BOOL;		//TRUE when link is OK on port A
	LinkOK_PortB											:	BOOL;		//TRUE when link is OK on port B - Redundancy port 

	{attribute 'displaymode':='hex'}  
	DevState										AT %I*	:	UINT; (*	Link to EtherCAT Master "DevState" under Inputs,
																				0x0001 = Link error
																				0x0002 = I/O locked after link error (I/O reset required)
																				0x0004 = Link error (redundancy adapter)
																				0x0008 = Missing one frame (redundancy mode)
																				0x0010 = Out of send resources (I/O reset required)
																				0x0020 = Watchdog triggered
																				0x0040 = Ethernet driver (miniport) not found
																				0x0080 = I/O reset active
																				0x0100 = At least one device in 'INIT' state
																				0x0200 = At least one device in 'PRE-OP' state
																				0x0400 = At least one device in 'SAFE-OP' state
																				0x0800 = At least one device indicates an error state
																				0x1000 = DC not in sync *)
	DevStateText											:	T_MAXSTRING;		//shows string of device state
	DevStateBits											:	EC_MASTER_DEVICE_STATE;
	DevStateChanged											:	BOOL; //TRUE if device state changed compared to previous cylce								
   	ResetRequired											:	BOOL;		//TRUE when a reset is requested
	MinOneSlaveNotInOP										:	BOOL;		//TRUE when at least one slave is available but not in OP state
    
	NoOfFrames												:	INT;		//No of frames configured
	FrmState										AT %I*	:	ARRAY [MIN_FRAMES..MAX_FRAMES] OF UINT;	//Link to EtherCAT Master "FrmStateXXX" under Inputs, e.g. 0x0001 = 1. EtherCAT command not sent (NOP requested)
	FrmWcState										AT %I*	:	ARRAY [MIN_FRAMES..MAX_FRAMES] OF UINT;	//Link to EtherCAT Master "FrmWcStateXXX" under Inputs, e.g. 0x0001 = wrong working counter of 1. EtherCAT command received
	FrmInputToggle									AT %I*	:	ARRAY [MIN_FRAMES..MAX_FRAMES] OF UINT;	//Link to EtherCAT Master "FrmInputToggleXXX" under Inputs, e.g. 0x0001 = Toggle Bit: 1. EtherCAT command received new inputs
	AllFramesMissing										:	BOOL;		//TRUE if all frames are missing 
	FramesWCState											:	BOOL;		//TRUE if WC state in at least one frame is <> 0
	FramesWcStateChanged									:	BOOL;		//TRUE if WC state of at least one frame changed compared to previous cylce	
	
	SlaveCount										AT %I*	:	UINT;	//Link to EtherCAT Master "SlaveCount" under Inputs, show actual numer of slaves 
	SlaveCount2										AT %I*	:	UINT;	//Link to EtherCAT Master "SlaveCount2" under Inputs, show actual numer of slaves in redunance mode
	SlaveCountTotal											:	UINT; 		//Slave count 1 and 2
	RedundanceActive										:	BOOL;		//Redundance active 		
            																				                    	
(* InfoData *)      	
	ChangeCount										AT %I*	:	UINT;					//Link to EtherCAT Master "ChangeCount" under InfoData, shows how often the image of content has changed
	DevId											AT %I*	:	UINT;					//Link to EtherCAT Master "DevId" under InfoData 
 	AmsNetId										AT %I*	:	ARRAY[0..5] OF BYTE; 	//Link to EtherCAT Master "AmsNetId" under InfoData
	AmsNetIdStr												:	T_AmsNetId;	//EtherCAT Master AmsNetId in string format
	CfgSlaveCount									AT %I*	:	UINT;					////Link to EtherCAT Master "CfgSlaveCount" under InfoData, reports configured no of EtherCAT slaves
         
(* DC timestamp *)
	DCTime													:	T_DCTIME64; // RealtimeTick in DC time 64, refreshed once per cycle*)             					
						
END_VAR

VAR
	MemDevState												:	UINT := 9999;	
	MemFrmWcState											:	ARRAY [MIN_FRAMES..MAX_FRAMES] OF UINT;	

	IOF_GetDeviceName										: 	IOF_GetDeviceName := (TMOUT	:= DEFAULT_ADS_TIMEOUT);
	EcMasterFrameCount										:	FB_EcMasterFrameCount := (tTimeout	:= DEFAULT_ADS_TIMEOUT);
	TON_LinkOK_PortA										:	TON := (PT := DELAY_LINK_OK);
	TON_LinkOK_PortB										:	TON := (PT := DELAY_LINK_OK);
	i														:	INT;
END_VAR

(* EcMaster IOs *)
DevStateChanged												:= DevState <> MemDevState;
IF DevStateChanged
THEN
	DevStateBits.NoError									:= DevState = 0;
	DevStateBits.LinkError 									:= DevState.0;
	DevStateBits.IOLockedAfterLinkError	    				:= DevState.1;
	DevStateBits.LinkErrorRedMode							:= DevState.2;
	DevStateBits.MissingOneFrmInRedMode     				:= DevState.3;
	DevStateBits.OutOfSendResources         				:= DevState.4;
	DevStateBits.WatchdogTriggered 		    				:= DevState.5;
	DevStateBits.EthernetDriverNotFound 					:= DevState.6;
	DevStateBits.IOResetActive 			    				:= DevState.7;
	DevStateBits.AtLeastOneSlaveInINIT      				:= DevState.8;
	DevStateBits.AtLeastOneSlaveInPREOP     				:= DevState.9;
	DevStateBits.AtLeastOneSlaveInSAFEOP    				:= DevState.10;
	DevStateBits.AtLeastOneSlaveInERROR     				:= DevState.11;																
	DevStateBits.DcNotInSync 		        				:= DevState.12;
	DevStateText 											:= F_ConvMasterDevStateToString(DevState);
	ResetRequired 											:= DevStateBits.IOLockedAfterLinkError OR DevStateBits.OutOfSendResources;
	MinOneSlaveNotInOP										:= DevStateBits.AtLeastOneSlaveInINIT OR DevStateBits.AtLeastOneSlaveInPREOP OR  DevStateBits.AtLeastOneSlaveInSAFEOP OR DevStateBits.AtLeastOneSlaveInERROR;
	MemDevState												:= DevState;
END_IF

RedundanceActive 											:= SlaveCount2 <> 0 AND SlaveCount <> 0;
SlaveCountTotal												:= SlaveCount2 + SlaveCount;

TON_LinkOK_PortA(IN:= NOT DevStateBits.LinkError 		, Q=> LinkOK_PortA );
TON_LinkOK_PortB(IN:= NOT DevStateBits.LinkErrorRedMode	, Q=> LinkOK_PortB );

AllFramesMissing 											:= TRUE;
FramesWCState												:= FALSE;	
FramesWcStateChanged										:= FALSE;
FOR i := MIN_FRAMES TO LIMIT(0,NoOfFrames -1, MAX_FRAMES) DO
	IF FrmWcState[i] <> 0 THEN
		FramesWCState										:= TRUE;
		IF FrmWcState[i].15 OR FrmWcState[i] = 16#7FFF THEN
			;
		ELSE
			AllFramesMissing 								:= FALSE;
		END_IF
	ELSE
		AllFramesMissing 									:= FALSE;
	END_IF
	
	IF MemFrmWcState[i] <> FrmWcState[i] 
	THEN
		FramesWcStateChanged								:= TRUE;
		MemFrmWcState[i]									:= FrmWcState[i]; 
	END_IF
END_FOR

//Get DC time 
DCTime														:= F_GetCurDcTickTime64();

(* Get Master Name *)
IF Name = ''
	AND DevId <> 0
	OR IOF_GetDeviceName.BUSY
	OR IOF_GetDeviceName.START
THEN
	AmsNetIdStr 											:= F_CreateAmsNetId(nIds := AmsNetId);
	IOF_GetDeviceName(
		NETID		:= '',
		DEVICEID	:= DevId,
		START		:= Name = '' AND NOT IOF_GetDeviceName.BUSY,
		TMOUT		:= ,
		BUSY		=> ,
		ERR			=> ,
		ERRID		=> ,
		DEVICENAME=> name);
END_IF

//No of config slaves 
IF EcMasterFrameCount.nFrames = 0
	AND DevId <> 0 
	OR EcMasterFrameCount.bBusy
	OR EcMasterFrameCount.bExecute
THEN
	EcMasterFrameCount(
		sNetId	:= AmsNetIdStr, 
		bExecute:= EcMasterFrameCount.nFrames = 0 AND NOT EcMasterFrameCount.bBusy, 
		tTimeout:= , 
		bBusy=> , 
		bError=> , 
		nErrId=> , 
		nFrames=> );
	NoOfFrames												:= TO_INT(EcMasterFrameCount.nFrames);
END_IF

(********************************************************************************************************)

END_FUNCTION_BLOCK

// ---- POUs/FileHandling/TF6421-XmlServer/XmlReadWriteWithBackupFile.TcPOU
{attribute 'no_check'}
//Write xml files with a additonal backup file and auto save function if structure will be changed.
//For the Backup functionality, a backup subfolder name "Backup" in the directory is needed! 
//In case the xml could not read successfully after, the backup files will be used.
//See Options to enable auto save and backup file functions.
//based on TF6421 - required lib: Tc2_XmlDataSvr - see Beckhoff documentation for more information
{attribute 'enable_dynamic_creation'}
FUNCTION_BLOCK XmlReadWriteWithBackupFile EXTENDS XmlReadWrite 
VAR_OUTPUT CONSTANT
{attribute 'displaymode':='binary'}
	OPTION_ENABLE_AUTO_SAVE									:	BYTE :=2#0000_0001;
{attribute 'displaymode':='binary'}
	OPTION_ENABLE_BACKUP_FILE								: 	BYTE :=2#0000_0010;
END_VAR                 									
VAR_INPUT               									                       		
{attribute 'displaymode':='binary'}
	Options													:	BYTE := 2#0000_0000;			(* option constants are alreay predefined, so they can accordingly be passed symbolically to the block 
																								Bit 0 = Enable auto save if data changed
																								Bit 1 = Enable backup file 
																								Bit 2 = 
																								Bit 3 = 
																								Bit 4 = 
																								Bit 5 = 
																								Bit 6 = 
																								Bit 7 = 						
																							*)     													
END_VAR
VAR_OUTPUT
	Backup													:	BOOL := FALSE; 		// Backup file has been readed 
	Loaded													:	BOOL:= FALSE;		// Data loaded
	ErrorFnc												:	STRING(30) := ''; 	// Error source
END_VAR
VAR
(* memory ************************************************************)
	rtExecuteAutoSave										:	R_trig;
	pCompareData											:	POINTER TO BYTE;
	pMemSymAddr												: 	PVOID := 0;	
	MemSymSize												:	UDINT;
(* Trigger **********************************************************)

(* timer ******************************************************************)
	tonDelay												:	ton;

(* function blocks ***************************************************************)

(* Dummy **********************************************************)

END_VAR

	(* XML Read/Write with backup file and auto save						V2.2		*)
	(************************************************************************************)

(* reserver memeory for auto save ***************************************************************************************)
	IF Options.0 AND pCompareData = 0 
	THEN	
		pCompareData 										:=  __NEW(BYTE, SymSize);
		IF NOT PARAM.ENABLE_DEBUG_MSG_DYNAMIC_MEM_ALLOCATION
		THEN 
			;
		ELSIF MemSymSize = 0 
		THEN
			AdsLogHint('EngineeringToolbox | FB XmlReadWriteWithBackupFile | An instance allocated %s bytes from the dynamic memory of the ADS router memory pool', TO_STRING(SymSize));	
		ELSE //Allocation of additional memory space
			AdsLogWarn('EngineeringToolbox | FB XmlReadWriteWithBackupFile | An instance allocated additional %s bytes from the dynamic memory of the ADS router memory pool because the size of the data increased (SymSize) ', TO_STRING(SymSize));
		END_IF
		MemSymSize											:= SymSize;
	ELSIF pCompareData <> 0 
	THEN
		IF NOT Options.0 OR SymSize > MemSymSize
		THEN //Delete pointer to allocated memory if no longer needed or size increase 
			__DELETE(pCompareData);
		ELSIF pMemSymAddr <> pSymAddr OR MemSymSize <> SymSize
		THEN //Erease data and rewrite if pointer to data changed or size decreased 
			MEMSET(pCompareData,0,MemSymSize); //Delete compare data if pointer to data changed to activate auto save
			MemSymSize										:= SymSize;
			pMemSymAddr 									:= pSymAddr;	
		END_IF
	END_IF
	
(* Execute sequence ***************************************************************************)	
	rtExecuteAutoSave(CLK := Options.0 AND state = 0 AND Loaded AND pCompareData <> 0 AND_THEN MEMCMP(pSymAddr, pCompareData, SymSize) <> 0);
	rtExecute(CLK := Execute );	
	
	CASE state OF
	0:
		Busy												:= FALSE;
		// init		                                	
		IF NOT Execute                              	
		THEN                                        	
			Backup											:= FALSE;			
			Done 											:= FALSE;
			Error											:= FALSE;
			ErrorID											:= 0;
			ErrorFnc										:= '';
		END_IF                                      	
		                                            	
		IF rtExecute.Q OR rtExecuteAutoSave.Q                       	
		THEN                                        	
			Backup											:= FALSE;
			Done 											:= FALSE;
			Busy											:= TRUE;
			Error											:= FALSE;
			ErrorID											:= 0;
			ErrorFnc										:= '';
			MemFnc											:= SEL(rtExecuteAutoSave.Q, Fnc, FNC_WRITE); // write has priority
			                                        	
			IF pSymAddr = 0                         	
			THEN                                    	
				Busy										:= NOT Error;
				Error										:= TRUE;
				ErrorId										:= E_AdsErr.DEVICE_INVALIDPARM;
				Done										:= FALSE;
				MemFnc										:= -1 ;
				RETURN;                             	
			ELSE
				CASE MemFnc OF
				FNC_READ:	
					XmlSrvRead	(bExecute := FALSE,sFilePath	:= CONCAT(FilePath,FileName));
					state 									:= 10;
				FNC_WRITE:	
					XmlSrvWrite	(bExecute := FALSE,sFilePath	:= CONCAT(FilePath,FileName));
					state 									:= 20;				
				ELSE
					Error									:= TRUE;
					ErrorID									:= E_AdsErr.DEVICE_INVALIDPARM;
					ErrorFnc								:= CONCAT('Invalid Fnc,', INT_TO_STRING(MemFnc));
					Busy									:= FALSE;			
				END_CASE
			END_IF
		END_IF
	
	(* File read ************************************************)
	10:
		XmlSrvRead(                    	
			sNetId		:= NetId,
			ePath		:= ,(* Default *)
			nMode		:= XMLSRV_SKIPMISSING, 
			pSymAddr	:= pSymAddr,
			cbSymSize	:= SymSize,
			sFilePath	:= ,
			sXPath		:= XPath,
			bExecute	:=  TRUE,
			tTimeout	:= Timeout,
			bBusy		=> ,
			bError		=> ,
			nErrId		=> );
			
		IF NOT XmlSrvRead.bBusy
		THEN
			IF XmlSrvRead.bError
			THEN
				IF XmlSrvRead.nErrId = 1804 
					AND Options.1
				THEN
					state									:= 11;
				ELSE
					Error									:= TRUE;
					ErrorID									:= XmlSrvRead.nErrId;
					ErrorFnc								:= CONCAT('XmlSvrRead State:',INT_TO_STRING(State));
					Busy									:= FALSE;
					State									:= 0;	
				END_IF
			ELSE
				Loaded										:= TRUE;
				Busy										:= FALSE;
				Done										:= TRUE;
				MemFnc										:= -1;
				state										:= 0;	
				IF pCompareData <> 0 THEN MEMCPY(pCompareData,pSymAddr,SymSize); pMemSymAddr := pSymAddr; END_IF 	// refresh compare data after reading for initalisation
			END_IF
			XmlSrvRead(bExecute 							:= FALSE);
		END_IF	
				
	11: // Read Backup file
		XmlSrvRead.sFilePath								:= CONCAT(FilePath,'Backup\'); 				// subfolder
		XmlSrvRead.sFilePath								:= CONCAT(XmlSrvRead.sFilePath,FileName);
				
		XmlSrvRead(                    	
			sNetId		:= NetId,
			ePath		:= ,(* Default *)
			nMode		:= XMLSRV_SKIPMISSING, 
			pSymAddr	:= pSymAddr,
			cbSymSize	:= SymSize,
			sFilePath	:= ,
			sXPath		:= XPath,
			bExecute	:=  TRUE,
			tTimeout	:= Timeout,
			bBusy		=> ,
			bError		=> ,
			nErrId		=> );
			
		IF NOT XmlSrvRead.bBusy
		THEN
			IF XmlSrvRead.bError
			THEN
				Error										:= TRUE;
				ErrorID										:= XmlSrvRead.nErrId;
				ErrorFnc									:= CONCAT('XmlSvrRead State:',INT_TO_STRING(State));
				Busy										:= FALSE;
				State										:= 0;	
			ELSE                                        	
				Loaded										:= TRUE;
				Backup										:= TRUE;
				Busy										:= FALSE;
				Done										:= TRUE;
				MemFnc										:= -1;
				state										:= 20; 							// Write original file	
				IF pCompareData <> 0 THEN MEMCPY(pCompareData,pSymAddr,SymSize); pMemSymAddr := pSymAddr; END_IF 	// refresh compare data after reading of backup file for initalisation
			END_IF
			XmlSrvRead(bExecute 							:= FALSE);
		END_IF	
		
	(* Write parameter ***********************************************************)
	20:
		XmlSrvWrite(
			sNetId		:= NetId,
			ePath		:= ,(* Default *)
			nMode		:= Mode,
			pSymAddr	:= pSymAddr,
			cbSymSize	:= SymSize,
			sFilePath	:= ,
			sXPath		:= XPath,
			bExecute	:= TRUE,
			tTimeout	:= Timeout,
			bBusy		=> ,
			bError		=> ,
			nErrId		=> );
			
		IF NOT XmlSrvWrite.bBusy
		THEN
			IF XmlSrvWrite.bError
			THEN
				Error										:= TRUE;
				ErrorID										:= XmlSrvWrite.nErrId;
				ErrorFnc									:= CONCAT('XmlSvrWrite State:',INT_TO_STRING(State));
				Busy										:= FALSE;
				State										:= 0;				
			ELSE // Write backup file	
				Loaded										:= TRUE;
				State										:= SEL(Options.1, 0, 21); //
				Done										:= State = 0; 				
				Busy										:= State <> 0;
				//Update compare memory
				IF pCompareData <> 0 THEN MEMCPY(pCompareData,pSymAddr,SymSize); pMemSymAddr := pSymAddr; END_IF 	// refresh compare data after writing new data
			END_IF
			XmlSrvWrite(bExecute							:= FALSE);
		END_IF

	21://Write backup to sub folder	
		XmlSrvWrite.sFilePath								:= CONCAT(FilePath,'Backup\'); 				// subfolder
		XmlSrvWrite.sFilePath								:= CONCAT(XmlSrvWrite.sFilePath,FileName);
		XmlSrvWrite(
			sNetId		:= NetId,
			ePath		:= ,(* Default *)
			nMode		:= Mode,
			pSymAddr	:= pSymAddr,
			cbSymSize	:= SymSize,
			sFilePath	:= ,
			sXPath		:= XPath,
			bExecute	:= TRUE,
			tTimeout	:= Timeout,
			bBusy		=> ,
			bError		=> ,
			nErrId		=> );
			
		IF NOT XmlSrvWrite.bBusy
		THEN
			IF XmlSrvWrite.bError
			THEN
				Error										:= TRUE;
				ErrorID										:= XmlSrvWrite.nErrId;
				ErrorFnc									:= CONCAT('XmlSvrWrite State:',INT_TO_STRING(State));
				Busy										:= FALSE;
				State										:= 0;				
			ELSE 	
				Busy										:= FALSE;
				Done										:= TRUE;
				State										:= 0;	
				//Update compare memory
				IF pCompareData <> 0 THEN MEMCPY(pCompareData,pSymAddr,SymSize); pMemSymAddr := pSymAddr; END_IF 	// refresh compare data after writing new data				
			END_IF
			XmlSrvWrite(bExecute							:= FALSE);
		END_IF		
	END_CASE
		
		
	
(*************************************************************************************************)

METHOD FB_exit : BOOL
VAR_INPUT
	bInCopyCode : BOOL; // if TRUE, the exit method is called for exiting an instance that is copied afterwards (online change).
END_VAR
IF NOT bInCopyCode AND pCompareData <> 0
THEN //Release memory in case the PLC stopps
	__DELETE(pCompareData);
END_IF
END_METHOD

PROPERTY PUBLIC optEnableAutoSave : BOOL
GET
optEnableAutoSave := Options.0;
END_GET
SET
Options.0 := optEnableAutoSave;
END_SET
END_PROPERTY

PROPERTY PUBLIC optEnableBackupFile : BOOL
GET
optEnableBackupFile := Options.1;
END_GET
SET
Options.1 := optEnableBackupFile;
END_SET
END_PROPERTY

METHOD PUBLIC read : BOOL //Return value = TRUE if busy
//required parameter
//pSymAddr
//SymSize
//FilePath
//XPath
VAR_INPUT
	Execute													:	BOOL;
END_VAR
CASE state OF
0:	
	Fnc 													:= FNC_READ;
	THIS^(Execute:=Execute);
1: 
	;

END_CASE
Read 														:= Busy;
END_METHOD

METHOD PUBLIC write : BOOL //Return value = TRUE if busy
//required parameter
//pSymAddr
//SymSize
//FilePath
//XPath
VAR_INPUT
	Execute													:	BOOL;
END_VAR
CASE state OF
0:	
	Fnc 													:= FNC_WRITE;
	THIS^(Execute:=Execute);
1: 
	;

END_CASE
Write 														:= Busy;
END_METHOD

END_FUNCTION_BLOCK

// ---- POUs/IO/Analog/AnalogInELMBase.TcPOU
// Based FB for analog input channels of ELM terminals incl. EtherCAT Slave Info Data 
//You can inherit your final implementation from this base "class"  
FUNCTION_BLOCK AnalogInELMBase EXTENDS EcSlaveInfoData
VAR_INPUT
	Enable													:	BOOL 	:= TRUE;
	MinValue												: 	LREAL 	:= 0.0;
	MaxValue												: 	LREAL 	:= 0.0;
	NoOfDigits												: 	INT 	(0..10)	:= 0; //number of decimal digits of scaled Q variable 
	OutOnError												:	LREAL 	:= 0.000000000000000001;
{attribute 'displaymode':='binary'}     	            	
	Options													:	BYTE  := 2#0000_0000;
END_VAR                 									
VAR                                     	            	
{attribute 'displaymode':='binary'}     	            	
	Status										AT  %I*		:	DWORD := 2#0100_0000_0000_0000;	//Terminal status (4 bytes) 
	
END_VAR                                 	            	
VAR_OUTPUT                              	            	                                       	
	(* Statusbist *)                    	
	NoOfSamples												:	USINT; //Byte 1
	Error													:	BOOL; //Byte2.0
	Underrange 												:	BOOL; //Byte2.1
	Overrange												:	BOOL ; //Byte2.2
	Diag													:	BOOL; //Byte2.4
	TxPDOState												:	BOOL; //Byte2.5
	InputCycleCounter										:	USINT; //Byte2.6/.7	
END_VAR                                 	
VAR                                     	
END_VAR

(* Base FB for ELM analog in terminals 																		*)
(************************************************************************************************************)

(* evaluate statusword **************************************************************************************)
	MEMCPY(ADR(NoOfSamples),ADR(Status),SIZEOF(NoOfSamples));
	Error													:= Enable AND (Status.8 OR MinValue = MaxValue AND NoOfDigits = 0);
	Underrange 												:= Status.9;
	Overrange												:= Status.10;
	
	Diag													:= Status.12;
	TxPDOState												:= Status.13; //True if not valid
	InputCycleCounter.0										:= Status.14;
	InputCycleCounter.1										:= Status.15;
	
(**********************************************************************************************************************)

END_FUNCTION_BLOCK

// ---- POUs/IO/Cylinder/Cylinder.TcPOU
{attribute 'no_check'}
//Cylinder object with two outputs (Workpos./Basepos) and correlated inputs
//Via the Options byte, it is possible to disable the use either of one or both feedback inputs.
//In case the physical feedback input in disabled, the status output of the FB will be generated by PT_Feedback
//In case the physical feedback input will not be triggerd to his corresonding outout within a certain time (PT_Feedback), an timeout error occures
//The physical outputs could be blocked by set the FeedxxxPos signals to false.
//FB "INPUT" is used inside
FUNCTION_BLOCK Cylinder IMPLEMENTS I_Cylinder
VAR_OUTPUT CONSTANT
{attribute 'displaymode':='binary'}
	OPTION_DISABLE_SENSOR_BASEPOS							:	BYTE  := 2#0000_0001; //Disable sensor check basepos. Feedback time used instead to create signal
{attribute 'displaymode':='binary'}
	OPTION_DISABLE_SENSOR_WORKPOS							:	BYTE  := 2#0000_0010; //Disable sensor check workpos. Feedback time used instead to create signal
{attribute 'displaymode':='binary'}
	OPTION_FREE												:	BYTE  := 2#0000_0100; //Not used option		
{attribute 'displaymode':='binary'}
	OPTION_DISABLE_LOGIC_ERROR								:	BYTE  := 2#0000_1000; //Disable logic error (Sensor workpos and basepos active at the same time) 	
{attribute 'displaymode':='binary'}
	OPTION_SWAP_SENSOR_STATUS								:	BYTE  := 2#0001_0000; //Swap signals work and base pos at Status byte
{attribute 'displaymode':='binary'}
	OPTION_INVERT_SENSOR_BASEPOS							:	BYTE  := 2#0010_0000; //Invert logic of sensor basepos (->NO)
{attribute 'displaymode':='binary'}
	OPTION_INVERT_SENSOR_WORKPOS							:	BYTE  := 2#0100_0000;//Invert logic of sensor workpos (->NO)
{attribute 'displaymode':='binary'}
	OPTION_EN_IMPULS_VALVE									:	BYTE  := 2#1000_0000; //Outputs are switched off if endposition is reached	
END_VAR
VAR_INPUT  (* Peripherie Outputs *)
	Quit													:	BOOL;	//Resets error with rising edge
	ToWorkPos												:	BOOL;	//moves cylinder to work position
	ToBasePos												:	BOOL;	//moves cylinder to base position
{attribute 'displaymode':='binary'}         			
	Options													:	BYTE  := 2#0000_0000;  (* option constants are predefined, so they can accordingly be passed symbolically to the block
																							DISABLE_FEEDBACK_BP	= .0
																							DISABLE_FEEDBACK_WP	= .1
																							ENABLE_LATCH_ERROR	= .2
																							DISABLE_LOGIC_ERROR	= .3																							
																							SWAP_SENSOR_STATUS	= .4
																							FEEDBACK_BP_INVERT	= .5
																							FEEDBACK_WP_INVERT	= .6
																							IMPULS_VALVE		= .7
																									*)
	FeedBasePos												:	BOOL := TRUE;	//enables feed in base direction
	FeedWorkPos												:	BOOL := TRUE;	//enables feed in work direction
	PT_Timeout												:	TIME := T#5S; 	//Runtime check BasePos
	PT_Feedback												:	TIME := T#3S; 	//Delay simulate Feedback
	PT_SensorDamping										:	TIME := T#0MS; 	//Work and Base pos sensor on/off damping time to suppress sensor flickering  
END_VAR                                     			
VAR_OUTPUT  (* Peripherie Inputs *)         			
	InBasePos												:	BOOL;	//TRUE when cylinder is in base position
	InWorkPos												:	BOOL;	//TRUE when cylinder is in work position
	Done													:	BOOL; 	//Limit sensor reached or feedback time counted down
	Busy													:	BOOL;	//Busy is TRUE at the rising edge of Execute and FALSE when one of the outputs Done, Aborted, or Error is set 
	ErrBasePos												:	BOOL;	//Cannot reach base position
	ErrWorkPos												:	BOOL;	//Cannot reach work position  
	ErrLogic												:	BOOL; 	//Both feedback signals are on
{attribute 'displaymode':='binary'}         			
	Status													:	BYTE;	(* 	Bit 0 = Q_ToBasePos or opposite if status swap in Options is active
																			Bit 1 = Q_ToWorkPos or opposite if status swap in Options is active
																			Bit 2 = InBasePos or opposite if status swap in Options is active
																			Bit 3 = InWorkPos or opposite if status swap in Options is active
																			Bit 4 = FeedBasePos or opposite if status swap in Options is active
																			Bit 5 = FeedWorkPos or opposite if status swap in Options is active
																			Bit 6 = Ready (no error)
																			Bit 7 = Error timeout move to position or sensor logic
																		*)
	Q_ToBasePos										AT  %Q* :	BOOL; //Hardware output - only with read access
	Q_ToWorkPos										AT  %Q* :	BOOL; //Hardware output - only with read access
END_VAR
VAR// IOs 
	SensorBasePos											: INPUT;
	SensorWorkPos											: INPUT;	
	TonErrBasePos											: TON;
	TonErrWorkPos											: TON;
	SimulationOn											:	BOOL;
END_VAR

	(* Cylinder	 IO V2.9					 								       	*)
	(* Includes functionblock "INPUT" 												*)
	(********************************************************************************)

(* Write Output *****************************************************)
	IF ToBasePos 	
	THEN
		moveToBasePos();
	ELSIF ToWorkPos AND NOT ToBasePos
	THEN
		moveToWorkPos();
	ELSE
		switchOff();
	END_IF

(* Reedkontakte lesen ***********************************************)
	this^._readSensors();
	
(* Status *************************************************)
	_writeStatus();
                        	
(* ack Error **********************************************************)
	IF Quit  THEN  reset(); END_IF

(* Timeout  ************************************************)
	_runtimeChk();
	
(*********************************************************************)

METHOD PROTECTED _readSensors : BOOL
VAR_INPUT
END_VAR
	SensorBasePos(
		Force	:= Q_ToBasePos AND NOT InWorkPos AND(Options.0 OR SimulationOn),
		Invert	:= Options.5,
		PT_ON	:= SEL(Options.0 OR SimulationOn,PT_SensorDamping,PT_FEEDBACK),
		PT_OFF	:= SEL(Options.0 OR SimulationOn,PT_SensorDamping,T#0MS),
		Q_DIRECT=>,
		Q		=> InBasePos,
		Q_RT	=> ,
		Q_FT	=> ,
		IN		=> );


	SensorWorkPos(
		Force	:= Q_ToWorkPos AND NOT InBasePos AND(Options.1 OR SimulationOn),
		Invert	:= Options.6,
		PT_ON	:= SEL(Options.1 OR SimulationOn ,PT_SensorDamping,PT_FEEDBACK),
		PT_OFF	:= SEL(Options.1 OR SimulationOn ,PT_SensorDamping,T#0MS),
		Q_DIRECT=>,
		Q		=> InWorkPos,
		Q_RT	=> ,
		Q_FT	=> ,
		IN		=> );
		

	_readSensors									:= TRUE;
END_METHOD

METHOD PROTECTED _runtimeChk : BOOL
VAR_INPUT
END_VAR
(* Timeout WorkPos ************************************************)
	TonErrWorkPos(	IN := Q_ToWorkPos AND (NOT InWorkPos OR InBasePos),
					PT := MAX(PT_Timeout + PT_SensorDamping,PT_Feedback + T#1S),
					Q => ErrWorkPos);

(* Timeout WorkPos ************************************************)
	tonErrBasePos(	IN := Q_ToBasePos AND (NOT InBasePos OR InWorkPos),
					PT := MAX(PT_Timeout + PT_SensorDamping,PT_Feedback + T#1S),
					Q => ErrBasePos);
					
(*********************************************************************)
	_runtimeChk									:= TRUE;
END_METHOD

METHOD PROTECTED _writeStatus : BOOL
VAR_INPUT
END_VAR


	(* Move *)
	IF Q_ToBasePos AND NOT Q_ToWorkPos AND (NOT InBasePos OR InWorkPos)
	THEN
		Status.0 											:= NOT Options.4;
		Status.1											:= Options.4;
	ELSIF Q_ToWorkPos AND NOT Q_ToBasePos AND (NOT InWorkPos OR InBasePos)
	THEN
		Status.0											:= Options.4;
		Status.1											:= NOT Options.4;
	END_IF              									

	(* BasePos / WorkPos reached*)
	Status.2 												:= SEL(Options.4, InBasePos , InWorkPos);
	Status.3 												:= SEL(Options.4, InWorkPos , InBasePos);
 				        									
	(* Feed ok *)    									
	Status.4 												:= SEL(Options.4, FeedBasePos , FeedWorkPos);
	Status.5 												:= SEL(Options.4, FeedWorkPos , FeedBasePos);
                        									
	(* Ready *)         									
	Status.6												:= NOT Status.7; 
	                    									
	(* Error *)         									
	Status.7 												:= ErrBasePos OR ErrWorkPos OR ErrLogic;
	
	(* Logic error bit **********************************************)
	ErrLogic												:= InBasePos AND InWorkPos AND NOT Options.3;
	
	(* Result *)
	_writeStatus												:= TRUE;
END_METHOD

METHOD PUBLIC enable : BOOL //Return Done = TRUE if WorkPos is TRUE and InWorkPos = TRUE or WorkPos is FALSE and InBasePos is TRUE 
VAR_INPUT
	IN													:	BOOL; //TRUE=WORK / FALSE=BASE
END_VAR
IF IN
THEN
	Enable 													:= THIS^.moveToWorkPos();
ELSE
	Enable 													:= This^.moveToBasePos();
END_IF
END_METHOD

{attribute 'monitoring' := 'call'}
PROPERTY PUBLIC inError : Bool
GET
InError									:= Status.7;
END_GET
END_PROPERTY

{attribute 'monitoring' := 'call'}
PROPERTY public isBusy : bool
GET
isBusy := Busy;
END_GET
END_PROPERTY

{attribute 'monitoring' := 'call'}
PROPERTY isInBasePos : BOOL
GET
isInBasePos := InBasePos;
END_GET
END_PROPERTY

{attribute 'monitoring' := 'call'}
PROPERTY isInWorkPos : BOOL
GET
isInWorkPos := InWorkPos;
END_GET
END_PROPERTY

{attribute 'monitoring' := 'call'}
PROPERTY public isOff : BOOL
GET
isOff := not ToWorkPos and not ToBasePos;
END_GET
END_PROPERTY

METHOD PUBLIC moveToBasePos : BOOL //Return = Done -> InBasePos
ToWorkPos 									:= Q_ToWorkPos	:= FALSE;
ToBasePos 													:= TRUE;
Q_ToBasePos	 												:= FeedBasePos AND (NOT Options.7 OR NOT InBasePos);
moveToBasePos 									:= Done			:= InBasePos;
Busy														:= NOT Done;
END_METHOD

METHOD PUBLIC moveToWorkPos : BOOL //Return = Done -> InWorkPos
ToBasePos 								:= Q_ToBasePos 		:= FALSE;
ToWorkPos													:= TRUE;
Q_ToWorkPos	 												:= FeedWorkPos AND (NOT Options.7 OR NOT InWorkPos);
moveToWorkPos								:= Done 				:= InWorkPos;
Busy														:= NOT Done;
END_METHOD

{attribute 'monitoring' := 'call'}
PROPERTY PUBLIC noFeed : BOOL
GET
noFeed						:= ToWorkPos and not FeedWorkPos or ToBasePos and not FeedBasePos;
END_GET
END_PROPERTY

{attribute 'monitoring' := 'call'}
PROPERTY Public ok : bool
GET
ok := Done;
END_GET
END_PROPERTY

{attribute 'monitoring' := 'call'}
PROPERTY PUBLIC optDisableLogicError : BOOL
GET
optDisableLogicError := Options.3;
END_GET
SET
Options.3 := optDisableLogicError;
END_SET
END_PROPERTY

{attribute 'monitoring' := 'call'}
PROPERTY PUBLIC optDisableSensorBasepos : BOOL
GET
optDisableSensorBasepos := Options.0;
END_GET
SET
OPtions.0 := optDisableSensorBasepos;
END_SET
END_PROPERTY

{attribute 'monitoring' := 'call'}
PROPERTY PUBLIC optDisableSensorWorkpos : BOOL
GET
optDisableSensorWorkpos := Options.1;
END_GET
SET
OPtions.1 := optDisableSensorWorkpos;
END_SET
END_PROPERTY

{attribute 'monitoring' := 'call'}
PROPERTY PUBLIC optEnableImpulsValveFnc : BOOL
GET
optEnableImpulsValveFnc := Options.7;
END_GET
SET
Options.7 := optEnableImpulsValveFnc;
END_SET
END_PROPERTY

{attribute 'monitoring' := 'call'}
PROPERTY PUBLIC optInvertSensorBasepos : BOOL
GET
optInvertSensorBasepos := Options.5;
END_GET
SET
Options.5 := optInvertSensorBasepos;
END_SET
END_PROPERTY

{attribute 'monitoring' := 'call'}
PROPERTY PUBLIC optInvertSensorWorkpos : BOOL
GET
optInvertSensorBasepos := Options.6;
END_GET
SET
Options.6 := optInvertSensorBasepos;
END_SET
END_PROPERTY

{attribute 'monitoring' := 'call'}
PROPERTY PUBLIC optSwapSensorStatus : BOOL
GET
optSwapSensorStatus := Options.4;
END_GET
SET
OPtions.4 := optSwapSensorStatus;
END_SET
END_PROPERTY

{attribute 'monitoring' := 'call'}
PROPERTY PUBLIC rCylinder : REFERENCE TO Cylinder
GET
rCylinder REF= This^;
END_GET
END_PROPERTY

METHOD PUBLIC reset : BOOL //Result = reset done
	TonErrWorkPos(IN := FALSE);
	tonErrBasePos(IN := FALSE);
	ErrWorkPos	:= ErrBasePos := ErrLogic						:= FALSE;										
	Status.7 													:= FALSE;
	reset														:= TRUE;
END_METHOD

{attribute 'monitoring' := 'call'}
PROPERTY simulation : BOOL
GET
simulation := SimulationOn;
END_GET
SET
SimulationOn := simulation;
END_SET
END_PROPERTY

METHOD PUBLIC switchOff : BOOL
VAR_INPUT
END_VAR
	ToWorkPos	:= FALSE;
	ToBasePos	:= FALSE;
	Done		:= FALSE;
	Busy		:= FALSE;
	Q_ToBasePos	:= FALSE;
	Q_ToWorkPos	:= FALSE;
	switchOff	:= TRUE;
END_METHOD

END_FUNCTION_BLOCK

// ---- POUs/IO/Input.TcPOU
{attribute 'no_check'}
FUNCTION_BLOCK Input
VAR_INPUT
	Force													:	BOOL := FALSE; 	//simulates Input
	Invert													:	BOOL := FALSE; 	//inverts the Hardware Input
	PT_ON													:	TIME := T#0MS;	//on delay
	PT_OFF													:	TIME := T#0MS;	//off delay
END_VAR             										
VAR_OUTPUT          										
	Q														:	BOOL;	//Signal Delay
	Q_RT													:	BOOL;	//R_Trig Signal of Q
	Q_FT													:	BOOL;	//F_Trig Signal of Q
	Q_DIRECT												:	BOOL; 	//Signal direct
	In												AT  %I* : 	BOOL; 	//Hardware Input
END_VAR
VAR
	TON														:	TON;
END_VAR

(* Input/Sensor Functionblock with On/Off	attenuation and rising / fallen edge 	V2.0	*)
(********************************************************************************************)

(************************************)
IF NOT Q THEN
	TON(IN := (IN OR Force) XOR Invert, PT := PT_ON);
	Q 														:= TON.Q;
	Q_RT 													:= Q;
	Q_FT 													:= FALSE;
	Q_DIRECT 												:= TON.IN;
ELSE
	TON(IN := NOT ((IN OR Force) XOR Invert), PT := PT_OFF);
	Q 														:= Q AND NOT TON.Q;
	Q_RT 													:= FALSE;
	Q_FT 													:= NOT Q;
	Q_DIRECT 												:= Q AND NOT TON.IN;
END_IF
(********************************************************************************************)

END_FUNCTION_BLOCK

// ---- POUs/IO/Cylinder/CylinderType4.TcPOU
{attribute 'no_check'}
//Cylinder with 2x inputs each for work and base position, extended from FB Cylinder
FUNCTION_BLOCK CylinderType4 EXTENDS Cylinder
VAR_OUTPUT CONSTANT
END_VAR
VAR_INPUT  
END_VAR                                     			
VAR_OUTPUT    
{attribute 'displaymode':='binary'}
	ErrInfo													:	BYTE; //.0 BP#1 | .1 BP#2 | .2 WP#1 | .3 WP#2 | .6 Logic Pair#1 | .7 Logic Pair#2 
END_VAR
VAR// IOs 
	SensorBasePos2											: INPUT;
	SensorWorkPos2											: INPUT;
END_VAR

	(* Cylinder	with two inputs for work and base pos each					      	*)
	(* Includes functionblock "INPUT" 												*)
	(********************************************************************************)

(* Write Output *****************************************************)
	IF ToBasePos 	
	THEN
		moveToBasePos();
	ELSIF ToWorkPos AND NOT ToBasePos
	THEN
		moveToWorkPos();
	ELSE
		switchOff();
	END_IF

(* Reedkontakte lesen ***********************************************)
	_readSensors();
	
(* Status *************************************************)
	_writeStatus();
                        	
(* ack Error **********************************************************)
	IF Quit  THEN  reset(); END_IF

(* Timeout  ************************************************)
	_runtimeChk();
	
(*********************************************************************)

METHOD PROTECTED _readSensors : BOOL
VAR_INPUT
END_VAR
(* Call super read sensors first *********************************)
	SUPER^._readSensors();

(* check inputs 2# ************************************************)
	SensorBasePos2(
		Force	:= SensorBasePos.Force ,
		Invert	:= SensorBasePos.Invert,
		PT_ON	:= SensorBasePos.PT_ON,
		PT_OFF	:= SensorBasePos.PT_OFF,
		Q_DIRECT=>,
		Q		=> ,
		Q_RT	=> ,
		Q_FT	=> ,
		IN		=> );


	SensorWorkPos2(
		Force	:= SensorWorkPos.Force,
		Invert	:= SensorWorkPos.Invert,
		PT_ON	:= SensorWorkPos.PT_ON,
		PT_OFF	:= SensorWorkPos.PT_OFF,
		Q_DIRECT=>,
		Q		=> ,
		Q_RT	=> ,
		Q_FT	=> ,
		IN		=> );
		
(* Write status ******************************************)
	InBasePos 									:= SensorBasePos.Q AND SensorBasePos2.Q;
	InWorkPos 									:= SensorWorkPos.Q AND SensorWorkPos2.Q;
	
(* Write error info ***************************************)
	ErrInfo.0									:= TonErrBasePos.Q AND NOT SensorBasePos.Q;
	ErrInfo.1									:= TonErrBasePos.Q AND NOT SensorBasePos2.Q;
	ErrInfo.2									:= TonErrWorkPos.Q AND NOT SensorBasePos.Q;
	ErrInfo.3									:= TonErrWorkPos.Q AND NOT SensorWorkPos2.Q;

	ErrInfo.6									:= SensorBasePos.Q AND SensorWorkPos.Q;
	ErrInfo.7									:= SensorBasePos2.Q AND SensorWorkPos2.Q;
	
(**************************************************************)
	_readSensors								:= TRUE;
	
(*****************************************************************)
END_METHOD

END_FUNCTION_BLOCK

// ---- POUs/IO/Drives/CoE/AxDriveCoE.TcPOU
{attribute 'no_check'}
//CoE Drive status and diagnosis
//Attention: "SwitchedOn" will be only true if bit 12 "FollowCmdValue" of statusword is used by drive
FUNCTION_BLOCK AxDriveCoE EXTENDS AxDriveBase     
VAR CONSTANT								
END_VAR                  						
VAR_INPUT                           						
	BrakeUnlock												:	BOOL := FALSE;
END_VAR
VAR_IN_OUT
END_VAR
VAR_OUTPUT
	BrakeUnlocked											:	BOOL;
	Status													:	CiA_DS402Statusword;	
	InfoData1										AT %I*	:	UINT;
	InfoData2										AT %I*	:	UINT;
END_VAR                             						
VAR
END_VAR
VAR
(* Cache *********************************************************************)

	// CoE Diagmessage
	StatusTrig												: BYTE;
	MemStatusTrig											: BYTE;
	
(* Timer ********************************************************************************)
  	readDiagDelay											: TON := (PT := T#50MS);
                                  						
(* Trigger ******************************************************************************)


(* Function blocks ****************************************************************************)
	ReadCoEDiagMsg											: EcCoEReadNewestDiagMsg := (Timeout := DEFAULT_ADS_TIMEOUT);	
	CoEWrite												: FB_EcCoeSdoWriteEx := (tTimeout := DEFAULT_ADS_TIMEOUT);	

(* Dummy Speicher **********************************************************)
END_VAR

	(* CoE Drive																		*)
	(************************************************************************************)

(* abort function-call if the reference is invalid *****************************)
IF NOT __ISVALIDREF(rAxis) 
THEN
	Fault													:= TRUE;
	SwitchedOn												:= FALSE;
	Ready													:= FALSE;
	RETURN;         										
END_IF

(* Call super class ****************************************************)
	SUPER^(); 
	
(* Read Statusword ********************************************************)	
	IF rAxis.Status.OpMode.SimulationAxis
	THEN
		IF rAxis.PlcToNc.ControlDWord.0
		THEN
			Status.readStatusword(TO_UINT(eCiA_DS402_STATUS_STATE.OPERATION_ENABLED));
		ELSE
			Status.readStatusword(TO_UINT(eCiA_DS402_STATUS_STATE.SWITCHED_ON));	
		END_IF
	ELSE
		Status.readStatusword(Statusword);
	END_IF			
	
	(* EL72xx DS402 Statusword
		Bit 0 : Ready to switch on
		Bit 1 : Switched on
		Bit 2 : Operation enabled
		Bit 3 : Fault
		Bit 4 : reserved
		Bit 5 : Quick stop (inverse)
		Bit 6 : Switch on disabled
		Bit 7 : Warning
		Bit 8 + 9 : reserved
		Bit 10 : TxPDOToggle (An-/Abwahl über 0x60DA)
		Bit 11 : Internal limit active
		Bit 12 : (drive follows command value)
		Bit 13 - 15 : reserved *)
		
(* DriveStatusBits ***********************************************)
	Fault													:= Status.Fault
																OR rAxis.NcToPlc.StateDWord.28 (* DriveDeviceError *)
																OR rAxis.NcToPlc.StateDWord.30; (* IODataInvalid *)
            												
	Ready 													:= NOT Fault
																AND(Status.ReadyToSwitchOn OR Status.SwitchedOn);

	SwitchedOn												:= Status.SwitchedOn AND NOT Fault;

	
(* manual override break ********************************************************)
	IF (BrakeUnlock XOR BrakeUnlocked)
		OR CoEWrite.bBusy
	THEN
		BrakeUnlocked										:= BrakeUnlock;
		CoEWrite(
			bExecute	:= NOT CoEWrite.bBusy AND NOT rAxis.NcToPlc.StateDWord.30 AND AdsAddr.port > 0 AND NOT rAxis.Status.OpMode.SimulationAxis,
			sNetId		:= F_CreateAmsNetId(nIds :=AdsAddr.netId),
			nSlaveAddr	:= AdsAddr.port, 
			nIndex		:= 16#8012, 
			nSubIndex	:= 16#1, 
			pSrcBuf		:= ADR(BrakeUnlocked), 
			cbBufLen	:= SIZEOF(BrakeUnlocked));
	END_IF
	
(* Read diagnoses ***********************************************************)
	StatusTrig.0											:= NOT Status.ReadyToSwitchOn;
	StatusTrig.1											:= Status.Fault;
	StatusTrig.2											:= Status.Warning AND NOT Status.Fault;
	
	CASE state OF
	0: // Read subindex of the newest diagnosis message
		
		readDiagDelay(IN := StatusTrig <> MemStatusTrig AND NOT rAxis.Status.OpMode.SimulationAxis AND AdsAddr.port > 0);
	
		IF readDiagDelay.Q
		THEN
			ReadCoEDiagMsg( Execute:= FALSE,  AdsAddr:= AdsAddr);
				
			IF NOT ReadCoEDiagMsg.Busy
			THEN
				MemStatusTrig 								:= StatusTrig; 
				readDiagDelay(IN := FALSE);			
				state 										:= state + 1;
			END_IF
		END_IF
	1: // read newest message
		ReadCoEDiagMsg( Execute:= TRUE,  AdsAddr:= AdsAddr);
		IF NOT ReadCoEDiagMsg.Busy
		THEN
			IF ReadCoEDiagMsg.Error
			THEN
				state										:= 0;
			ELSE	
				state										:= 0;			
			END_IF
			ReadCoEDiagMsg(Execute := FALSE);		
		END_IF
		
	END_CASE
	
(******************************************************************************)

END_FUNCTION_BLOCK

// ---- POUs/IO/Drives/CoE/CiA_DS402Statusword.TcPOU
FUNCTION_BLOCK CiA_DS402Statusword
VAR_INPUT
END_VAR
VAR_OUTPUT	
	ReadyToSwitchOn			: BOOL; //Bit 0: Ready TO switch on	- - Controlled by state machine
	SwitchedOn				: BOOL; //Bit 1: Switched on - Controlled by state machine
	OperationEnabled		: BOOL; //Bit 2: Operation enabled - Controlled by state machine
	Fault					: BOOL; //Bit 3: Drive fault active
	VoltageEnabled			: BOOL; //Bit 4 - Manufacturer specific / Voltage enabled
	QuickStopInverse		: BOOL; // Bit 5: False = Quick stop active (inverse signal)- Controlled by state machine
	SwitchOnDisabled		: BOOL; // Bit 6: Switch in disabled - Controlled by state machine
	Warning					: BOOL; // Bit 7: Warning active
//Manufacturer specific_Bit8
	RemoteActive			: BOOL;  // Bit 9: ManufacturerSpecific_Bit9, commonly used for control over network (EtherCAT) active
//	TargetReached			: BOOL; // Bit 10 commonly used for in target position, velocity in pp or pv mode
//	TxPDOToggle				: BOOL; // Bit 10: TxPDOToggle (An-/Abwahl über 0x8010:01)
	InternalLimitActive		: BOOL; // Bit 11: Internal limit active
//Operation mode specific_Bit12	- pp = Set-point acknowledge, pv = standstill, hm = Homing attained, csp = following set pos., csv following set velo
//Operation mode specific_Bit13 - pp = Following error, pv = N/A, hm = Homing error, csp = Following error, csv = N/A
//Manufacturer specific_Bit14
//Manufacturer specific_Bit15

	State					: eCiA_DS402_STATUS_STATE; // Device state
END_VAR

METHOD PUBLIC readStatusword : BOOL
VAR_INPUT
	Statusword 					:	UINT;
END_VAR
//Status bits
ReadyToSwitchOn												:= Statusword.0 ;
SwitchedOn													:= Statusword.1 ;
OperationEnabled											:= Statusword.2 ;
Fault														:= Statusword.3 ;
VoltageEnabled												:= Statusword.4 ;
QuickStopInverse											:= Statusword.5 ;
SwitchOnDisabled											:= Statusword.6 ;
Warning														:= Statusword.7 ;

RemoteActive												:= Statusword.9 ;

InternalLimitActive											:= Statusword.11;


//State
IF NOT ReadyToSwitchOn 
THEN
	IF SwitchOnDisabled
	THEN
		state												:= eCiA_DS402_STATUS_STATE.SWITCH_ON_DISABLED;
	ELSE
		state												:= eCiA_DS402_STATUS_STATE.NOT_READY_TO_SWITCH_ON;
	END_IF
ELSIF Fault
THEN
	IF ReadyToSwitchOn AND SwitchedOn AND OperationEnabled
	THEN
		state												:= eCiA_DS402_STATUS_STATE.FAULT_REACTION_ACTIVE;
	ELSE
		state												:= eCiA_DS402_STATUS_STATE.FAULT_ACTIVE;
	END_IF
ELSE 
	IF QuickStopInverse
	THEN
		state												:= eCiA_DS402_STATUS_STATE.READY_TO_SWITCH_ON;
		IF SwitchedOn
		THEN
			state											:= eCiA_DS402_STATUS_STATE.SWITCHED_ON;
			IF OperationEnabled
			THEN
				state										:= eCiA_DS402_STATUS_STATE.OPERATION_ENABLED;
			END_IF
		END_IF
	ELSE //Quick stop active
		IF SwitchedOn AND OperationEnabled
		THEN
			state											:= eCiA_DS402_STATUS_STATE.QUICK_STOP_ACTIVE;
		ELSIF SwitchOnDisabled
		THEN
			state											:= eCiA_DS402_STATUS_STATE.SWITCH_ON_DISABLED;
		ELSE
			state 											:= eCiA_DS402_STATUS_STATE.NOT_READY_TO_SWITCH_ON;
		END_IF
	END_IF
END_IF

readStatusword												:= TRUE;
END_METHOD

END_FUNCTION_BLOCK

// ---- POUs/IO/Drives/CoE/EL72xx/AxDriveCoE_EL72xxParam.TcPOU
{attribute 'no_check'}
//FB template to read and write parameter
//The FB can be enherided and derivatived methods of SeqRead/SeqWrite used for application specific parameter.
//The extended methods need to call the super class at the beginning and return true if execution will be finished. The allowed states for new parameter are 1..99
FUNCTION_BLOCK AxDriveCoE_EL72xxParam EXTENDS AxRWParaBase
VAR_OUTPUT CONSTANT
END_VAR                                 					
VAR_INPUT                               					
	AdsAddr													: 	AMSADDR; //Terminal AMS Net Addr.     
	Channel													:	USINT := 0; //Drive channel 0 or 1                                    	                                        	
	SetKvPosition											:	LREAL; //(rad/s)rad - e.g. 10.0		0x8010:17
	SetKpVelocity											:	LREAL; //mA/(rad/s) - e.g. 0.058	0x8010:15
	SetTnVelocity											:	LREAL; //0.1ms 		- e.g. 0.015	0x8010:14
END_VAR 
VAR_IN_OUT
END_VAR                               					
VAR_OUTPUT
	DeviceType												:	STRING(15); //0x1008:0 -e.g. EL7211-9014
	MotorSN													:	STRING(15); //0x9009:13 - if available
	KvPosition												:	LREAL;
	KpVelocity												:	LREAL;
	TnVelocity												:	LREAL;	
END_VAR                         	
VAR
(* Cache ************************************************************)

(* Trigger **********************************************************)

(* Timer ******************************************************************)

(* FBs ***************************************************************)
	CoEWrite												: FB_EcCoESdoWriteEx := (tTimeout := DEFAULT_ADS_TIMEOUT); //CoE read
	CoERead													: FB_EcCoeSdoReadEx := (tTimeout := DEFAULT_ADS_TIMEOUT);

(* Dummy memory **********************************************************)
END_VAR

	(* Read/Write drive parameter														*)
	(************************************************************************************)

(* Execute ***************************************************************************************)
	SUPER^();

(*************************************************************************************************)

PROPERTY PROTECTED deviceAddrIsValid : BOOL
GET
deviceAddrIsValid := AdsAddr.port > 0;
END_GET
END_PROPERTY

METHOD PROTECTED getValue : BOOL //Return value = TRUE if execution finished and state incremented 
VAR_INPUT
	Index						:	WORD;
	SubIndex					:	BYTE;
	Len							:	UDINT;
	pActValue					:	PVOID; //Address of variable for actual value
	pSetValue					:	PVOID; //Address of variable for ser value variable, can be zero if no corresponding SetVariable exists
	CompleteAccess				:	BOOL;
END_VAR
CoERead(bExecute := TRUE , nIndex := Index ,nSubIndex := SubIndex ,pDstBuf := pActValue ,cbBufLen := Len, bCompleteAccess  := CompleteAccess);
IF NOT CoERead.bBUSY 	
THEN
	IF NOT CoERead.bError
	THEN
		IF pSetValue <> 0 THEN MEMCPY(pSetValue, pActValue, Len); END_IF
		state 												:= state + 1; 
	ELSE
		Busy												:= FALSE;
		Error												:= TRUE;
		ErrorId												:= CoERead.nErrId;
		ErrorText											:= CONCAT('Error read parameter in state:' , TO_STRING(state * -1));
		ErrorText											:= CONCAT(ErrorText , ' Id:');
		ErrorText											:= CONCAT(ErrorText , TO_STRING(ErrorId));
		State												:= 9999;
	END_IF
	CoERead(bExecute := FALSE);
	getValue												:= TRUE;
END_IF
END_METHOD

METHOD PROTECTED seqRead : BOOL //Return value = TRUE if execution finished 
VAR_IN_OUT
	state							:	INT;
END_VAR

(* Sequence read parameter **********************************)
	CASE state OF
	1..99: //Read application specific parameter  
		SeqRead												:= TRUE;
		
	1001: (* Init step ******************************************************)
		CoERead(bExecute := FALSE, sNetId:= F_CreateAmsNetId(nIds := AdsAddr.netId), nSlaveAddr:= AdsAddr.port);
		IF NOT CoERead.bBusy
		THEN
			state											:= state + 1;	
		END_IF
		
	1002: (* Device name *************************************************************************************)
		IF LEN(DeviceType) > 0 AND NOT CoERead.bBusy
		THEN
			state											:= state + 1;
		ELSE
			getValue(Index:= 16#1008,	Subindex := 16#0,	LEN := SIZEOF(DeviceType),	pActValue := ADR(DeviceType),	pSetValue := 0, completeAccess := FALSE);
		END_IF

	1003: (* Motor SN *************************************************************************************)		
		IF LEN(MotorSN) > 0 AND NOT CoERead.bBusy
		THEN
			state											:= state + 1;
		ELSE
			getValue(Index:= 16#9009,	Subindex := 16#03,	LEN := SIZEOF(MotorSN),		pActValue := ADR(MotorSN),	pSetValue := 0, completeAccess := FALSE);
		END_IF
			
	1004: (* kv position *******************************************)
		IF getValue(Index:= 16#8010,	Subindex := 16#17,	LEN := SIZEOF(_UDINT),		pActValue := ADR(_UDINT),	pSetValue := 0, completeAccess := FALSE)
		THEN
			KvPosition := SetKvPosition						:= SEL(Error, TO_LREAL(_UDINT) * 1.0, 0.0); 
		END_IF
	
	1005: (* Kp velocity *******************************************)
		IF getValue(Index:= 16#8010,	Subindex := 16#15,	LEN := SIZEOF(_UDINT),		pActValue := ADR(_UDINT),	pSetValue := 0, completeAccess := FALSE)
		THEN
			KpVelocity := SetKpVelocity						:= SEL(Error, TO_LREAL(_UDINT) * 0.001, 0.0);
		END_IF
		
	1006: (* Tn velocity ********************************************)
		IF getValue(Index:= 16#8010,	Subindex := 16#14,	LEN := SIZEOF(_UDINT),		pActValue := ADR(_UDINT),	pSetValue := 0, completeAccess := FALSE)
		THEN
			TnVelocity := SetTnVelocity						:= SEL(Error, TO_LREAL(_UDINT) * 0.0001, 0.0);
		END_IF
	ELSE
		state												:= 1;
	END_CASE

(***********************************************************************************)
END_METHOD

METHOD PROTECTED seqWrite : BOOL //Return value = TRUE if execution finished 
VAR_IN_OUT
	state							:	INT;
END_VAR
(* Sequence write parameter *********************************************)
	CASE state OF
	1..99: //Write application specific parameter  
		SeqWrite											:= TRUE;
		
	1001: (* Init step ******************************************************)
		CoEWrite(bExecute := FALSE, sNetId:= F_CreateAmsNetId(nIds := AdsAddr.netId), nSlaveAddr:= AdsAddr.port);
		IF NOT CoEWrite.bBusy
		THEN
			state											:= state + 1;	
		END_IF
	
	1002: (* Kv position *************************************************************************************)
		_UDINT												:= TO_UDINT(SetKvPosition * 1.0);
		IF setValue(Index:= 16#8010,	Subindex := 16#17,	LEN := SIZEOF(_UDINT),		pActValue := 0,		pSetValue := ADR(_UDINT) , completeAccess := FALSE)
		THEN
			KvPosition										:= SetKvPosition;
		END_IF
		
	1003: (* Kp velocity ****************************************)
		_UDINT											:= TO_UDINT(SetKpVelocity * 1000.0);
		IF setValue(Index:= 16#8010,	Subindex := 16#15,	LEN := SIZEOF(_UDINT),		pActValue := 0,		pSetValue := ADR(_UDINT), completeAccess := FALSE)
		THEN
			KpVelocity										:= SetKpVelocity;
		END_IF

	1004: (* Tn velocity **********************************)
		_UDINT											:= TO_UDINT(SetTnVelocity * 10000.0);
		IF setValue(Index:= 16#8010,	Subindex := 16#14,	LEN := SIZEOF(_UDINT),		pActValue := 0,		pSetValue := ADR(_UDINT), completeAccess := FALSE)
		THEN
			TnVelocity										:= SetTnVelocity;
		END_IF	
	ELSE
		state												:= 1;
	END_CASE

(************************************************************************************)
END_METHOD

METHOD PROTECTED setValue : BOOL //Return value = TRUE if execution finished and state incremented 
VAR_INPUT
	Index						:	Word;
	SubIndex					:	BYTE;
	Len							:	UDINT;
	pActValue					:	PVOID; //Address of variable for actual value, can be zero if no corresponding acual value variable exists
	pSetValue					:	PVOID; //Address of variable for set value variable
	CompleteAccess				:	BOOL;
END_VAR


